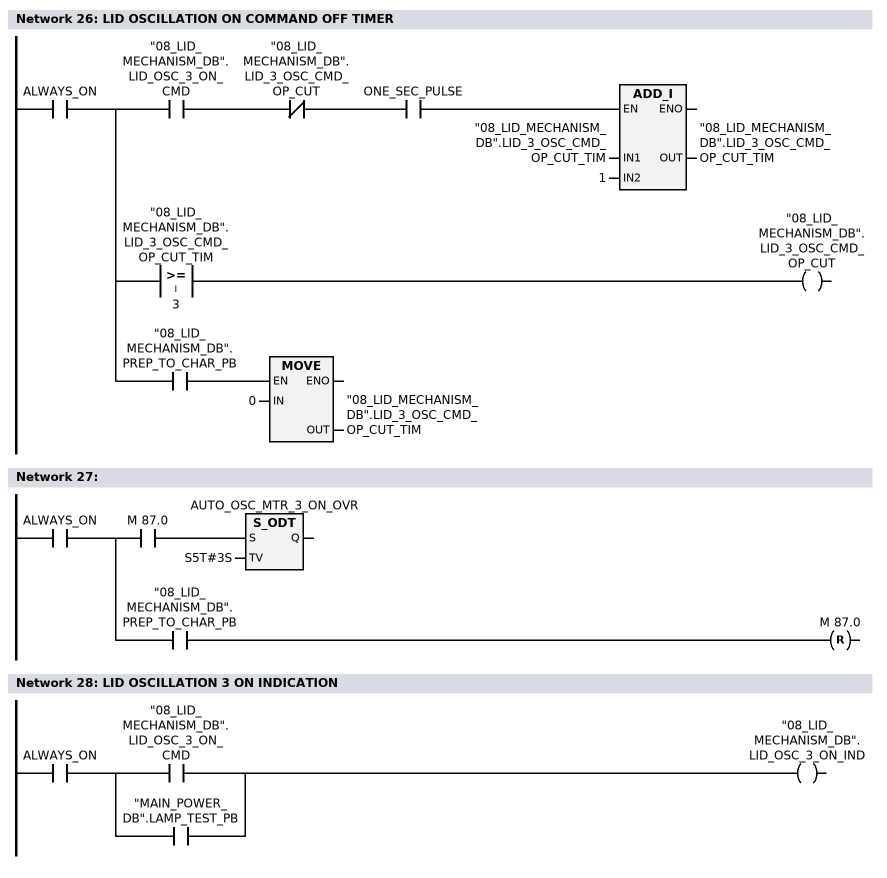
[picture p192: LID_3_MECHANISM networks 26-28]
NETWORK
TITLE = LID OSCILLATION ON COMMAND OFF TIMER
      A     "ALWAYS_ON";
      =     L 0.0;
      A     L 0.0;
      A     "08_LID_MECHANISM_DB".LID_OSC_3_ON_CMD;
      AN    "08_LID_MECHANISM_DB".LID_3_OSC_CMD_OP_CUT;
      A     "ONE_SEC_PULSE";
      JNB   _00d;
      L     "08_LID_MECHANISM_DB".LID_3_OSC_CMD_OP_CUT_TIM;
      L     1;
      +I;
      T     "08_LID_MECHANISM_DB".LID_3_OSC_CMD_OP_CUT_TIM;
_00d: NOP   0;
      A     L 0.0;
      A(;
      L     "08_LID_MECHANISM_DB".LID_3_OSC_CMD_OP_CUT_TIM;
      L     3;
      >=I;
      );
      =     "08_LID_MECHANISM_DB".LID_3_OSC_CMD_OP_CUT;
      A     L 0.0;
      A     "08_LID_MECHANISM_DB".PREP_TO_CHAR_PB;
      JNB   _00e;
      L     0;
      T     "08_LID_MECHANISM_DB".LID_3_OSC_CMD_OP_CUT_TIM;
_00e: NOP   0;
NETWORK
TITLE =
      A     "ALWAYS_ON";
      =     L 0.0;
      A     L 0.0;
      A     M 87.0;
      L     S5T#3S;
      SD    "AUTO_OSC_MTR_3_ON_OVR";
      NOP   0;
      NOP   0;
      NOP   0;
      NOP   0;
      A     L 0.0;
      A     "08_LID_MECHANISM_DB".PREP_TO_CHAR_PB;
      R     M 87.0;
NETWORK
TITLE = LID OSCILLATION 3 ON INDICATION
//CHECK IT
      A     "ALWAYS_ON";
      A(;
      O     "08_LID_MECHANISM_DB".LID_OSC_3_ON_CMD;
      O     "MAIN_POWER_DB".LAMP_TEST_PB;
      );
      =     "08_LID_MECHANISM_DB".LID_OSC_3_ON_IND;
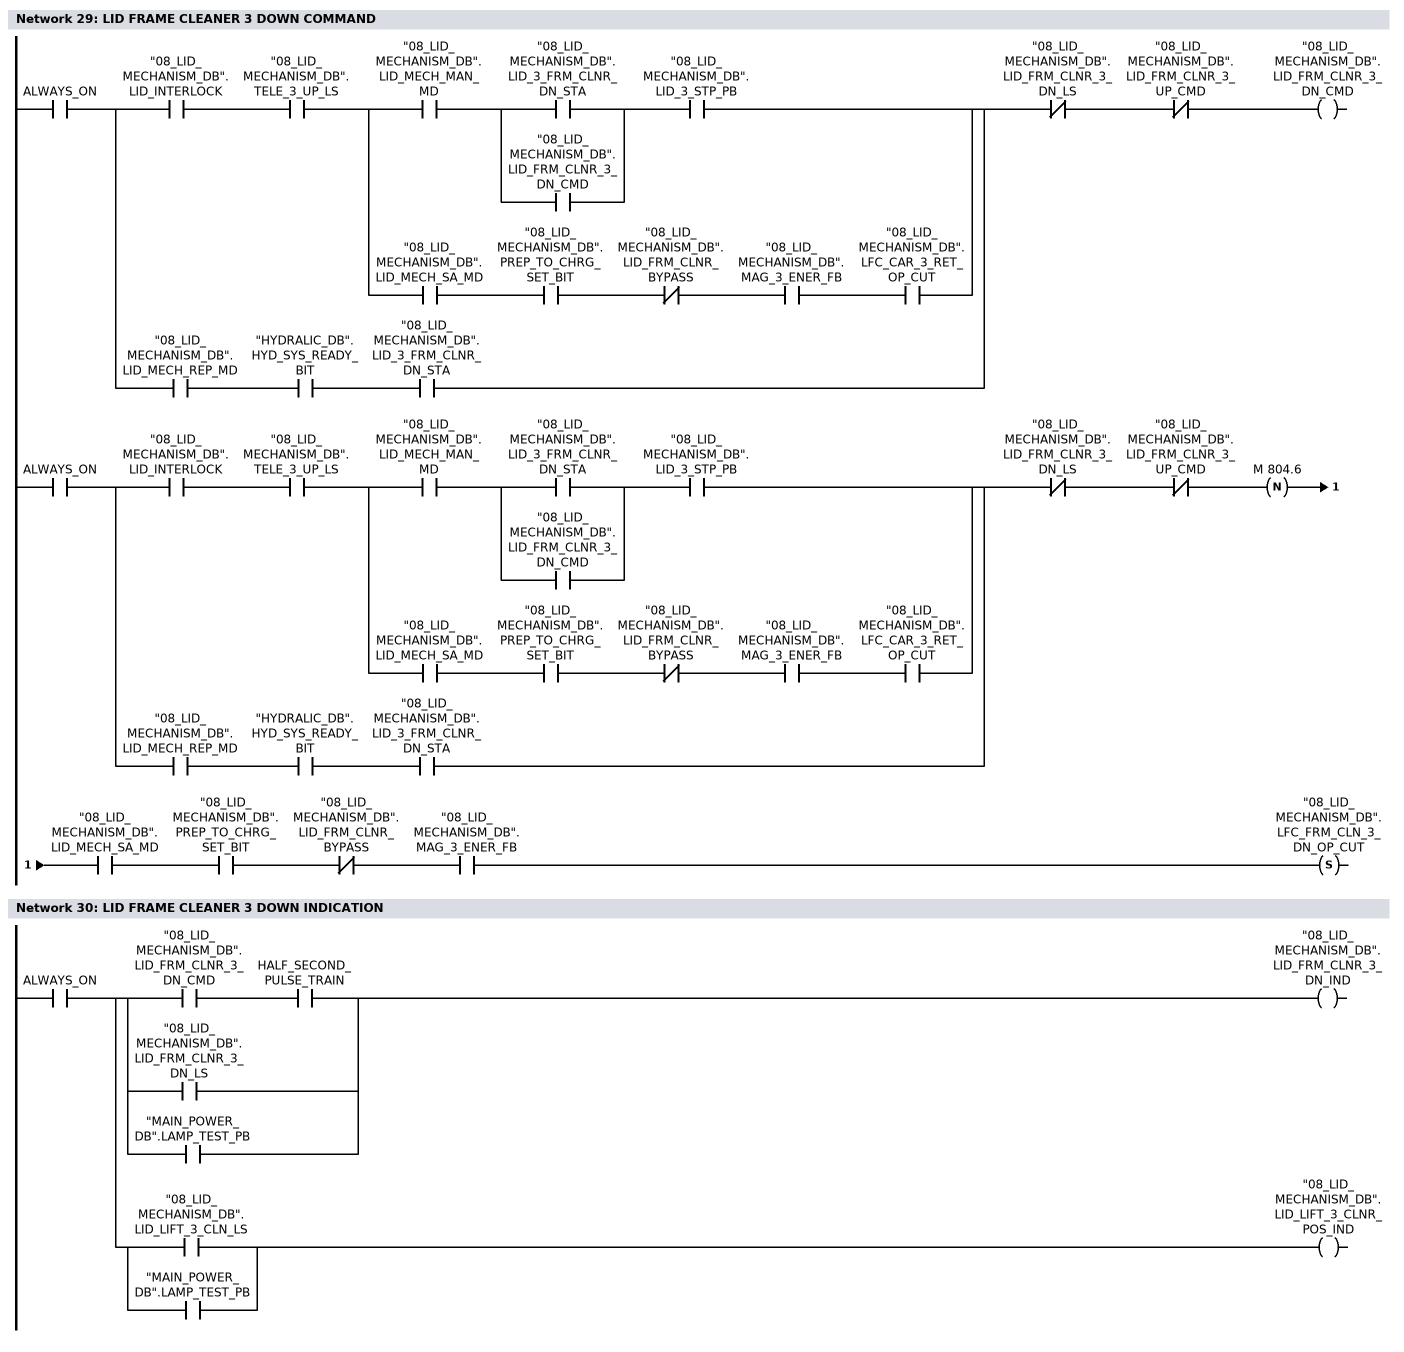
NETWORK
TITLE = LID FRAME CLEANER 3 DOWN COMMAND
      A     "ALWAYS_ON";
      A(;
      A     "08_LID_MECHANISM_DB".LID_INTERLOCK;
      A     "08_LID_MECHANISM_DB".TELE_3_UP_LS;
      A(;
      A     "08_LID_MECHANISM_DB".LID_MECH_MAN_MD;
      A(;
      O     "08_LID_MECHANISM_DB".LID_3_FRM_CLNR_DN_STA;
      O     "08_LID_MECHANISM_DB".LID_FRM_CLNR_3_DN_CMD;
      );
      A     "08_LID_MECHANISM_DB".LID_3_STP_PB;
      O;
      A     "08_LID_MECHANISM_DB".LID_MECH_SA_MD;
      A     "08_LID_MECHANISM_DB".PREP_TO_CHRG_SET_BIT;
      AN    "08_LID_MECHANISM_DB".LID_FRM_CLNR_BYPASS;
      A     "08_LID_MECHANISM_DB".MAG_3_ENER_FB;
      A     "08_LID_MECHANISM_DB".LFC_CAR_3_RET_OP_CUT;
      );
      O;
      A     "08_LID_MECHANISM_DB".LID_MECH_REP_MD;
      A     "HYDRALIC_DB".HYD_SYS_READY_BIT;
      A     "08_LID_MECHANISM_DB".LID_3_FRM_CLNR_DN_STA;
      );
      AN    "08_LID_MECHANISM_DB".LID_FRM_CLNR_3_DN_LS;
      AN    "08_LID_MECHANISM_DB".LID_FRM_CLNR_3_UP_CMD;
      =     L 0.0;
      A     L 0.0;
      BLD   102;
      =     "08_LID_MECHANISM_DB".LID_FRM_CLNR_3_DN_CMD;
      A(;
      A     L 0.0;
      FN    M 804.6;
      );
      A     "08_LID_MECHANISM_DB".LID_MECH_SA_MD;
      A     "08_LID_MECHANISM_DB".PREP_TO_CHRG_SET_BIT;
      AN    "08_LID_MECHANISM_DB".LID_FRM_CLNR_BYPASS;
      A     "08_LID_MECHANISM_DB".MAG_3_ENER_FB;
      S     "08_LID_MECHANISM_DB".LFC_FRM_CLN_3_DN_OP_CUT;
NETWORK
TITLE = LID FRAME CLEANER 3 DOWN INDICATION
      A     "ALWAYS_ON";
      =     L 0.0;
      A     L 0.0;
      A(;
      A     "08_LID_MECHANISM_DB".LID_FRM_CLNR_3_DN_CMD;
      A     "HALF_SECOND_PULSE_TRAIN";
      O     "08_LID_MECHANISM_DB".LID_FRM_CLNR_3_DN_LS;
      O     "MAIN_POWER_DB".LAMP_TEST_PB;
      );
      =     "08_LID_MECHANISM_DB".LID_FRM_CLNR_3_DN_IND;
      A     L 0.0;
      A(;
      O     "08_LID_MECHANISM_DB".LID_LIFT_3_CLN_LS;
      O     "MAIN_POWER_DB".LAMP_TEST_PB;
      );
      =     "08_LID_MECHANISM_DB".LID_LIFT_3_CLNR_POS_IND;
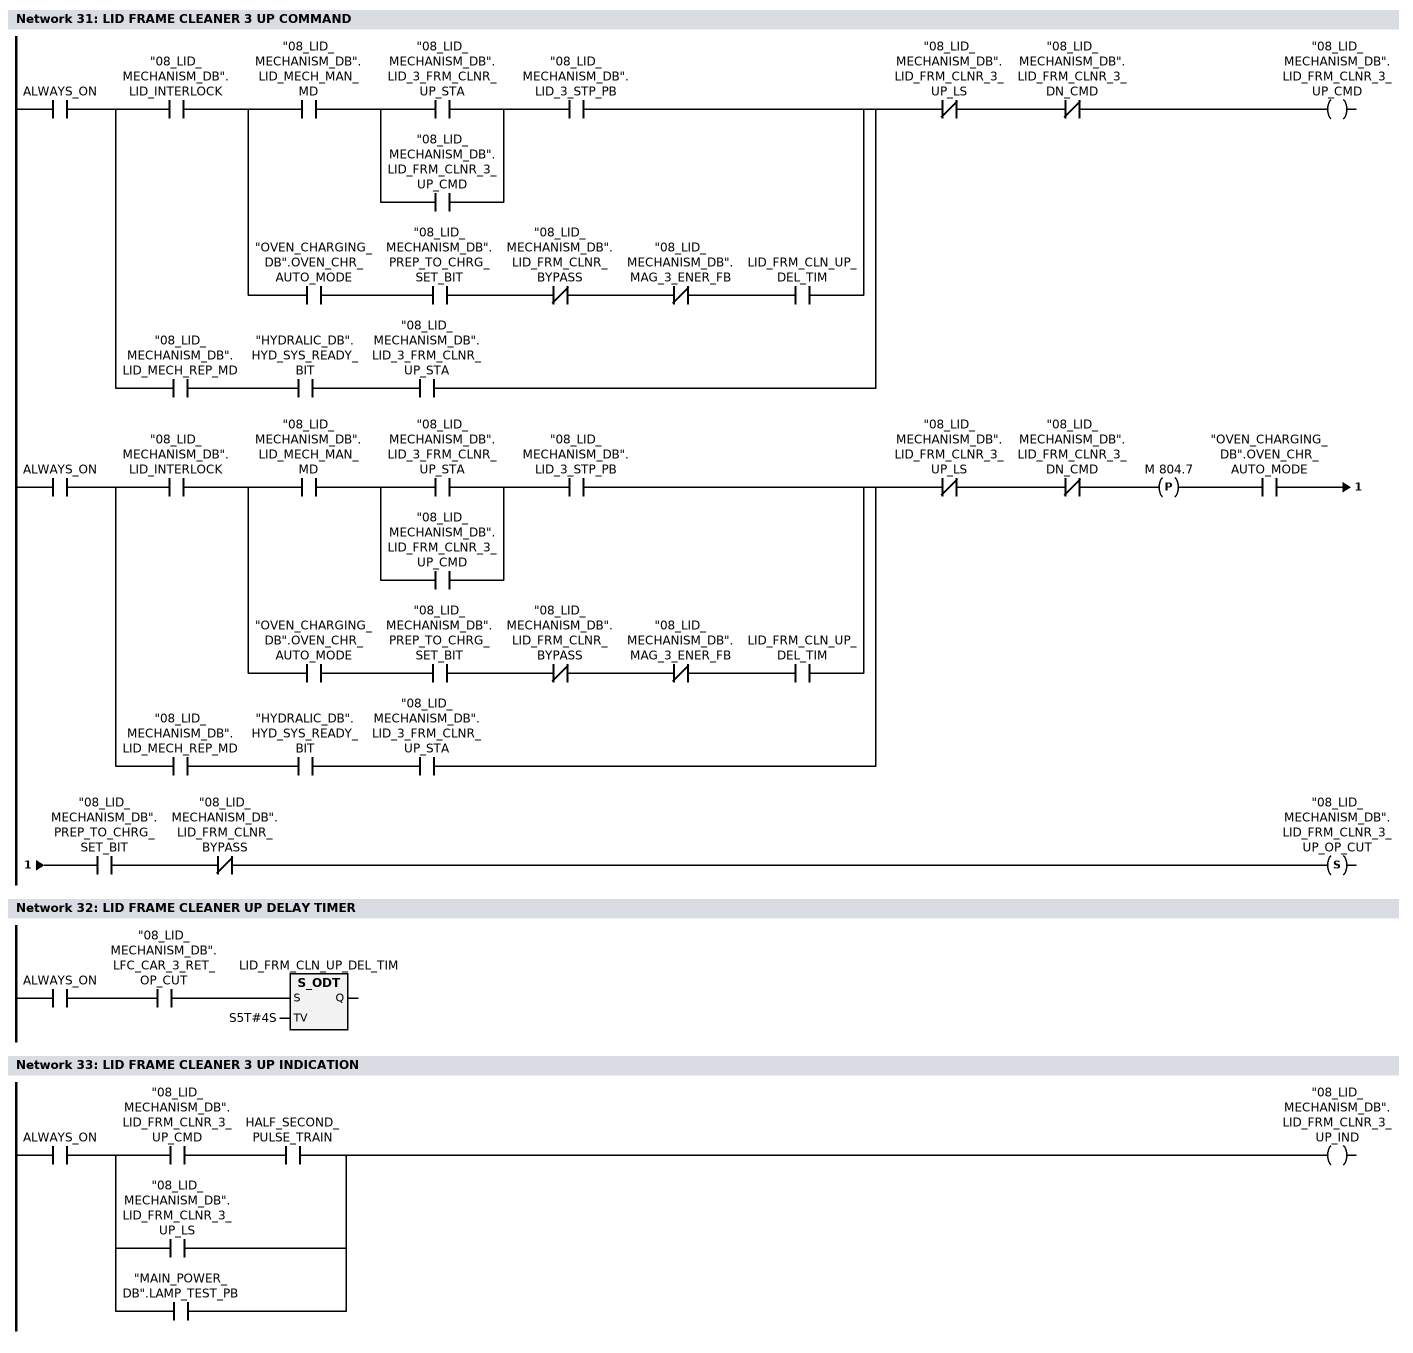
NETWORK
TITLE = LID FRAME CLEANER 3 UP COMMAND
      A     "ALWAYS_ON";
      A(;
      A     "08_LID_MECHANISM_DB".LID_INTERLOCK;
      A(;
      A     "08_LID_MECHANISM_DB".LID_MECH_MAN_MD;
      A(;
      O     "08_LID_MECHANISM_DB".LID_3_FRM_CLNR_UP_STA;
      O     "08_LID_MECHANISM_DB".LID_FRM_CLNR_3_UP_CMD;
      );
      A     "08_LID_MECHANISM_DB".LID_3_STP_PB;
      O;
      A     "OVEN_CHARGING_DB".OVEN_CHR_AUTO_MODE;
      A     "08_LID_MECHANISM_DB".PREP_TO_CHRG_SET_BIT;
      AN    "08_LID_MECHANISM_DB".LID_FRM_CLNR_BYPASS;
      AN    "08_LID_MECHANISM_DB".MAG_3_ENER_FB;
      A     "LID_FRM_CLN_UP_DEL_TIM";
      );
      O;
      A     "08_LID_MECHANISM_DB".LID_MECH_REP_MD;
      A     "HYDRALIC_DB".HYD_SYS_READY_BIT;
      A     "08_LID_MECHANISM_DB".LID_3_FRM_CLNR_UP_STA;
      );
      AN    "08_LID_MECHANISM_DB".LID_FRM_CLNR_3_UP_LS;
      AN    "08_LID_MECHANISM_DB".LID_FRM_CLNR_3_DN_CMD;
      =     L 0.0;
      A     L 0.0;
      BLD   102;
      =     "08_LID_MECHANISM_DB".LID_FRM_CLNR_3_UP_CMD;
      A(;
      A     L 0.0;
      FP    M 804.7;
      );
      A     "OVEN_CHARGING_DB".OVEN_CHR_AUTO_MODE;
      A     "08_LID_MECHANISM_DB".PREP_TO_CHRG_SET_BIT;
      AN    "08_LID_MECHANISM_DB".LID_FRM_CLNR_BYPASS;
      S     "08_LID_MECHANISM_DB".LID_FRM_CLNR_3_UP_OP_CUT;
NETWORK
TITLE = LID FRAME CLEANER UP DELAY TIMER
      A     "ALWAYS_ON";
      A     "08_LID_MECHANISM_DB".LFC_CAR_3_RET_OP_CUT;
      L     S5T#4S;
      SD    "LID_FRM_CLN_UP_DEL_TIM";
      NOP   0;
      NOP   0;
      NOP   0;
      NOP   0;
NETWORK
TITLE = LID FRAME CLEANER 3 UP INDICATION
      A     "ALWAYS_ON";
      A(;
      A     "08_LID_MECHANISM_DB".LID_FRM_CLNR_3_UP_CMD;
      A     "HALF_SECOND_PULSE_TRAIN";
      O     "08_LID_MECHANISM_DB".LID_FRM_CLNR_3_UP_LS;
      O     "MAIN_POWER_DB".LAMP_TEST_PB;
      );
      =     "08_LID_MECHANISM_DB".LID_FRM_CLNR_3_UP_IND;
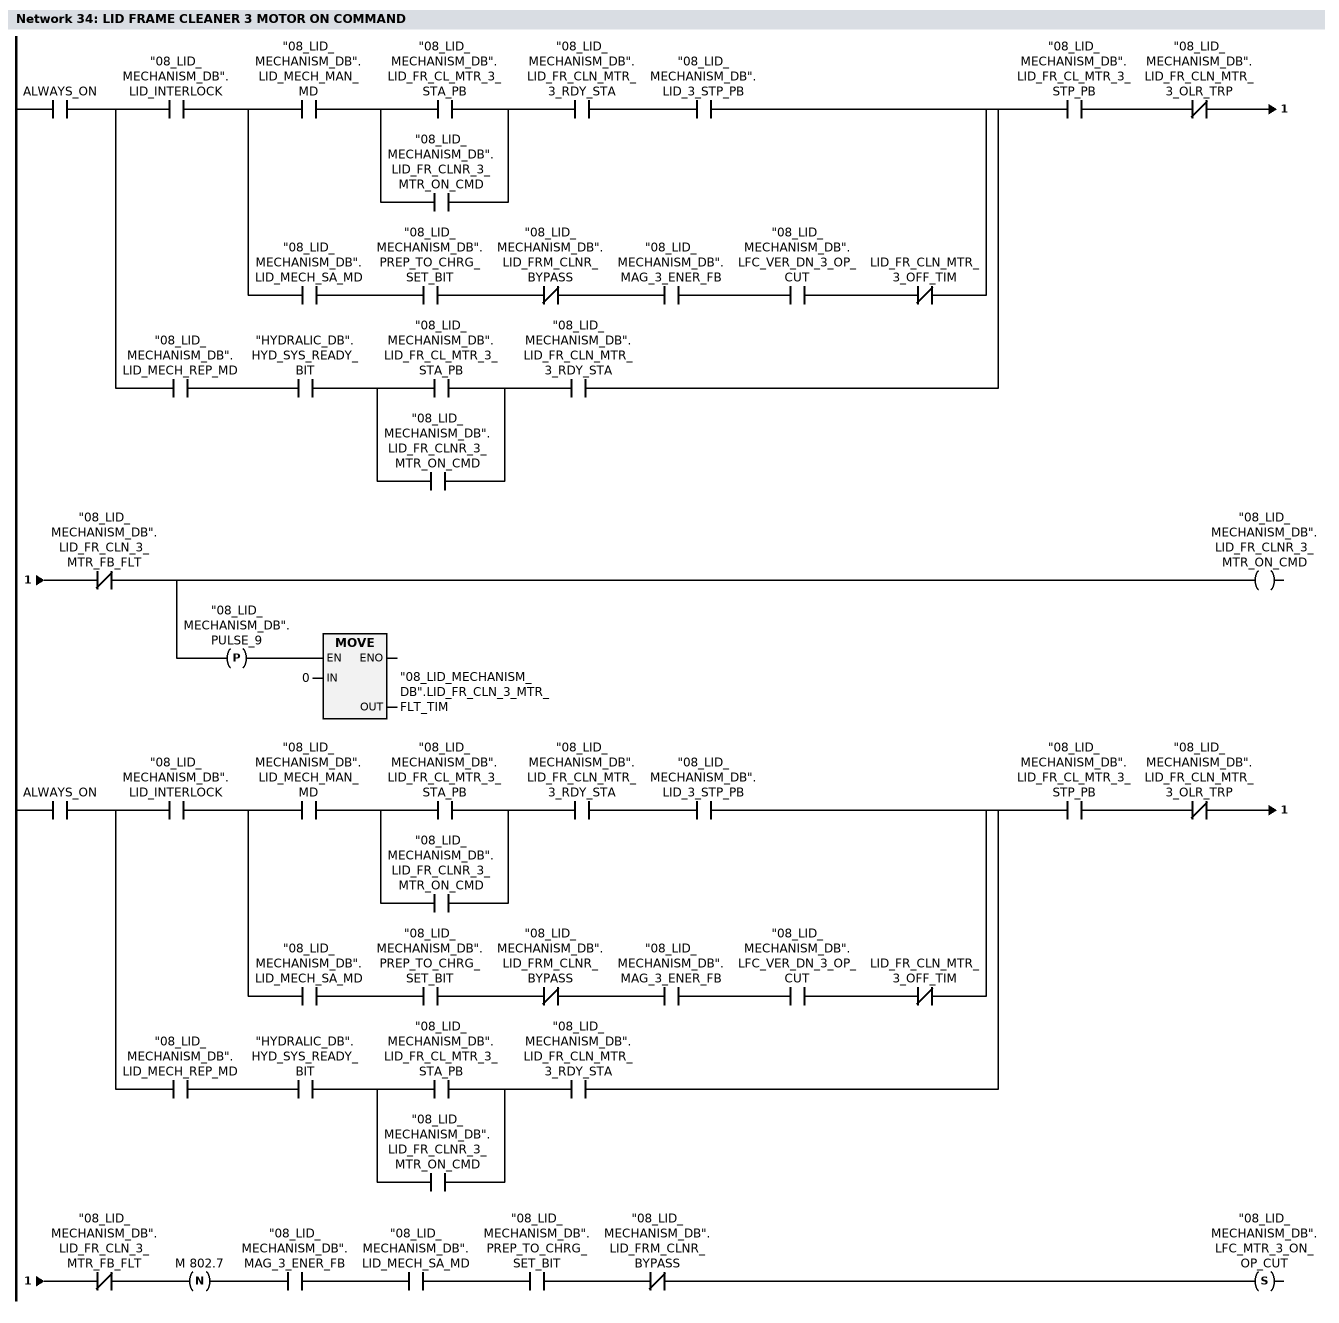
NETWORK
TITLE = LID FRAME CLEANER 3 MOTOR ON COMMAND
      A     "ALWAYS_ON";
      A(;
      A     "08_LID_MECHANISM_DB".LID_INTERLOCK;
      A(;
      A     "08_LID_MECHANISM_DB".LID_MECH_MAN_MD;
      A(;
      O     "08_LID_MECHANISM_DB".LID_FR_CL_MTR_3_STA_PB;
      O     "08_LID_MECHANISM_DB".LID_FR_CLNR_3_MTR_ON_CMD;
      );
      A     "08_LID_MECHANISM_DB".LID_FR_CLN_MTR_3_RDY_STA;
      A     "08_LID_MECHANISM_DB".LID_3_STP_PB;
      O;
      A     "08_LID_MECHANISM_DB".LID_MECH_SA_MD;
      A     "08_LID_MECHANISM_DB".PREP_TO_CHRG_SET_BIT;
      AN    "08_LID_MECHANISM_DB".LID_FRM_CLNR_BYPASS;
      A     "08_LID_MECHANISM_DB".MAG_3_ENER_FB;
      A     "08_LID_MECHANISM_DB".LFC_VER_DN_3_OP_CUT;
      AN    "LID_FR_CLN_MTR_3_OFF_TIM";
      );
      O;
      A     "08_LID_MECHANISM_DB".LID_MECH_REP_MD;
      A     "HYDRALIC_DB".HYD_SYS_READY_BIT;
      A(;
      O     "08_LID_MECHANISM_DB".LID_FR_CL_MTR_3_STA_PB;
      O     "08_LID_MECHANISM_DB".LID_FR_CLNR_3_MTR_ON_CMD;
      );
      A     "08_LID_MECHANISM_DB".LID_FR_CLN_MTR_3_RDY_STA;
      );
      A     "08_LID_MECHANISM_DB".LID_FR_CL_MTR_3_STP_PB;
      AN    "08_LID_MECHANISM_DB".LID_FR_CLN_MTR_3_OLR_TRP;
      AN    "08_LID_MECHANISM_DB".LID_FR_CLN_3_MTR_FB_FLT;
      =     L 0.0;
      A     L 0.0;
      BLD   102;
      =     "08_LID_MECHANISM_DB".LID_FR_CLNR_3_MTR_ON_CMD;
      A     L 0.0;
      FP    "08_LID_MECHANISM_DB".PULSE_9;
      JNB   _00f;
      L     0;
      T     "08_LID_MECHANISM_DB".LID_FR_CLN_3_MTR_FLT_TIM;
_00f: NOP   0;
      A(;
      A     L 0.0;
      FN    M 802.7;
      );
      A     "08_LID_MECHANISM_DB".MAG_3_ENER_FB;
      A     "08_LID_MECHANISM_DB".LID_MECH_SA_MD;
      A     "08_LID_MECHANISM_DB".PREP_TO_CHRG_SET_BIT;
      AN    "08_LID_MECHANISM_DB".LID_FRM_CLNR_BYPASS;
      S     "08_LID_MECHANISM_DB".LFC_MTR_3_ON_OP_CUT;
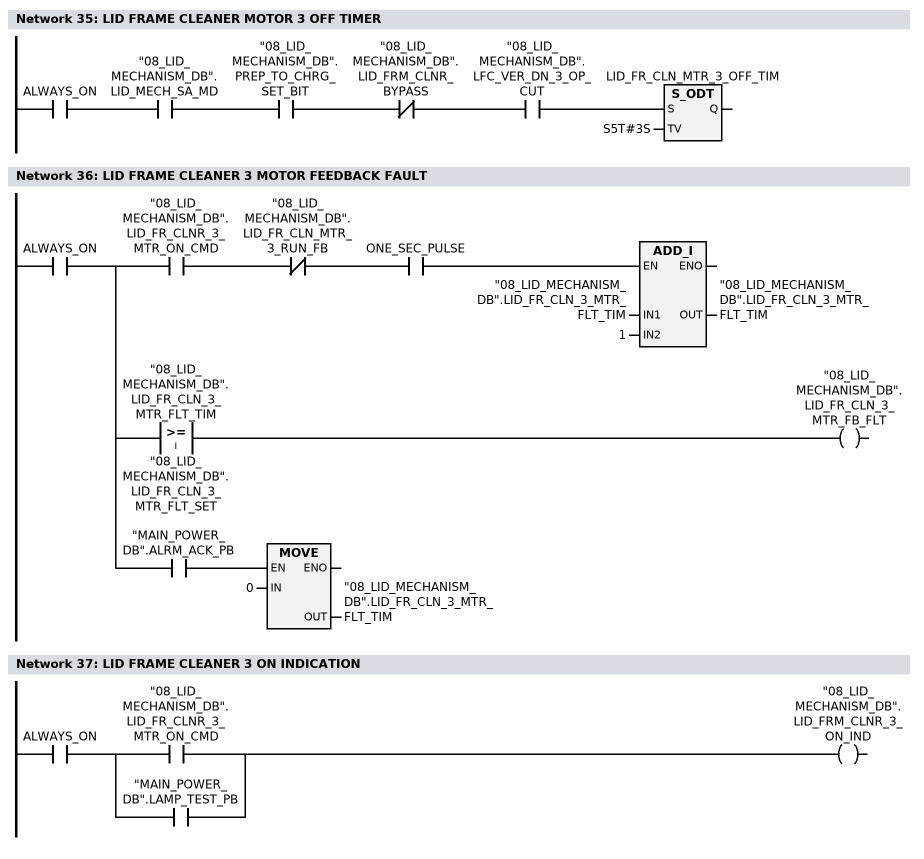
NETWORK
TITLE = LID FRAME CLEANER MOTOR 3 OFF TIMER
      A     "ALWAYS_ON";
      A     "08_LID_MECHANISM_DB".LID_MECH_SA_MD;
      A     "08_LID_MECHANISM_DB".PREP_TO_CHRG_SET_BIT;
      AN    "08_LID_MECHANISM_DB".LID_FRM_CLNR_BYPASS;
      A     "08_LID_MECHANISM_DB".LFC_VER_DN_3_OP_CUT;
      L     S5T#3S;
      SD    "LID_FR_CLN_MTR_3_OFF_TIM";
      NOP   0;
      NOP   0;
      NOP   0;
      NOP   0;
NETWORK
TITLE = LID FRAME CLEANER 3 MOTOR FEEDBACK FAULT
      A     "ALWAYS_ON";
      =     L 0.0;
      A     L 0.0;
      A     "08_LID_MECHANISM_DB".LID_FR_CLNR_3_MTR_ON_CMD;
      AN    "08_LID_MECHANISM_DB".LID_FR_CLN_MTR_3_RUN_FB;
      A     "ONE_SEC_PULSE";
      JNB   _010;
      L     "08_LID_MECHANISM_DB".LID_FR_CLN_3_MTR_FLT_TIM;
      L     1;
      +I;
      T     "08_LID_MECHANISM_DB".LID_FR_CLN_3_MTR_FLT_TIM;
_010: NOP   0;
      A     L 0.0;
      A(;
      L     "08_LID_MECHANISM_DB".LID_FR_CLN_3_MTR_FLT_TIM;
      L     "08_LID_MECHANISM_DB".LID_FR_CLN_3_MTR_FLT_SET;
      >=I;
      );
      =     "08_LID_MECHANISM_DB".LID_FR_CLN_3_MTR_FB_FLT;
      A     L 0.0;
      A     "MAIN_POWER_DB".ALRM_ACK_PB;
      JNB   _011;
      L     0;
      T     "08_LID_MECHANISM_DB".LID_FR_CLN_3_MTR_FLT_TIM;
_011: NOP   0;
NETWORK
TITLE = LID FRAME CLEANER 3 ON INDICATION
      A     "ALWAYS_ON";
      A(;
      O     "08_LID_MECHANISM_DB".LID_FR_CLNR_3_MTR_ON_CMD;
      O     "MAIN_POWER_DB".LAMP_TEST_PB;
      );
      =     "08_LID_MECHANISM_DB".LID_FRM_CLNR_3_ON_IND;
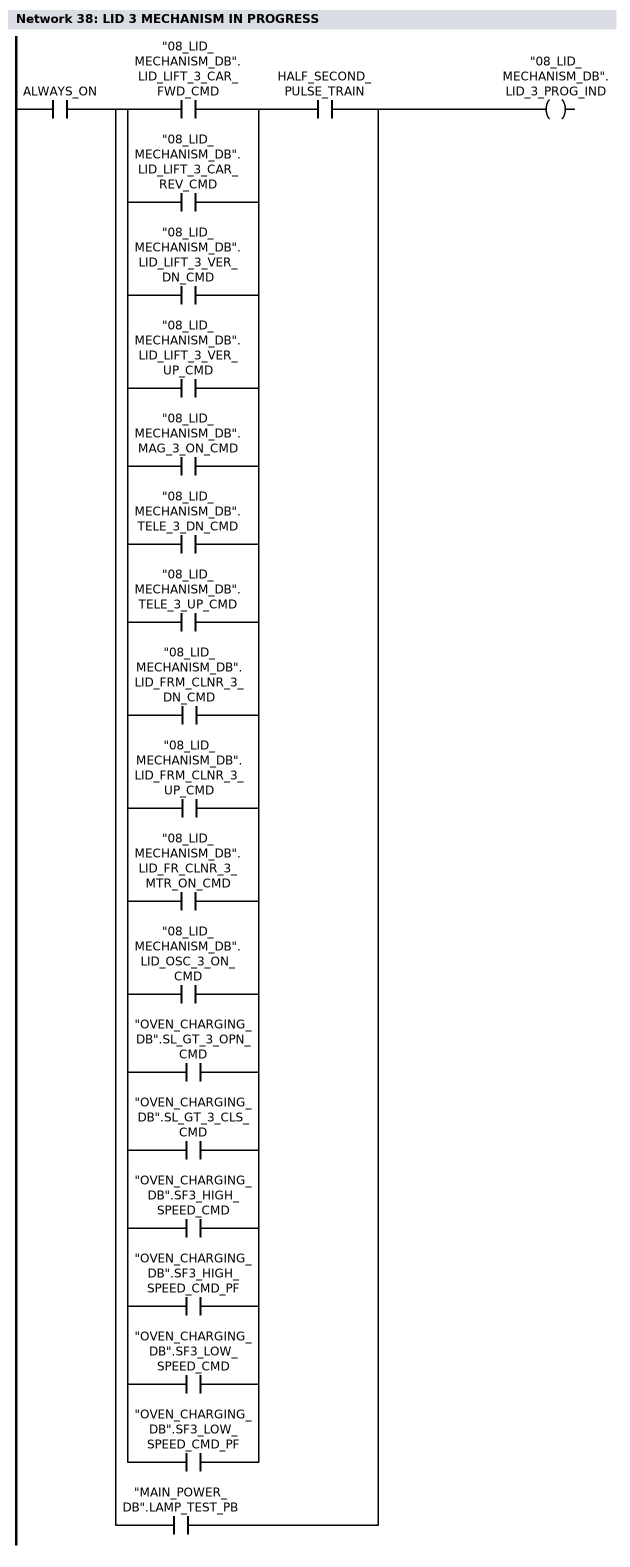
NETWORK
TITLE = LID 3 MECHANISM IN PROGRESS
      A     "ALWAYS_ON";
      A(;
      A(;
      O     "08_LID_MECHANISM_DB".LID_LIFT_3_CAR_FWD_CMD;
      O     "08_LID_MECHANISM_DB".LID_LIFT_3_CAR_REV_CMD;
      O     "08_LID_MECHANISM_DB".LID_LIFT_3_VER_DN_CMD;
      O     "08_LID_MECHANISM_DB".LID_LIFT_3_VER_UP_CMD;
      O     "08_LID_MECHANISM_DB".MAG_3_ON_CMD;
      O     "08_LID_MECHANISM_DB".TELE_3_DN_CMD;
      O     "08_LID_MECHANISM_DB".TELE_3_UP_CMD;
      O     "08_LID_MECHANISM_DB".LID_FRM_CLNR_3_DN_CMD;
      O     "08_LID_MECHANISM_DB".LID_FRM_CLNR_3_UP_CMD;
      O     "08_LID_MECHANISM_DB".LID_FR_CLNR_3_MTR_ON_CMD;
      O     "08_LID_MECHANISM_DB".LID_OSC_3_ON_CMD;
      O     "OVEN_CHARGING_DB".SL_GT_3_OPN_CMD;
      O     "OVEN_CHARGING_DB".SL_GT_3_CLS_CMD;
      O     "OVEN_CHARGING_DB".SF3_HIGH_SPEED_CMD;
      O     "OVEN_CHARGING_DB".SF3_HIGH_SPEED_CMD_PF;
      O     "OVEN_CHARGING_DB".SF3_LOW_SPEED_CMD;
      O     "OVEN_CHARGING_DB".SF3_LOW_SPEED_CMD_PF;
      );
      A     "HALF_SECOND_PULSE_TRAIN";
      O     "MAIN_POWER_DB".LAMP_TEST_PB;
      );
      =     "08_LID_MECHANISM_DB".LID_3_PROG_IND;
END_FUNCTION

FUNCTION "TATA_COMMUNICATION" : VOID	// FC 21
AUTHOR : Arun
VERSION : 0.1
BEGIN
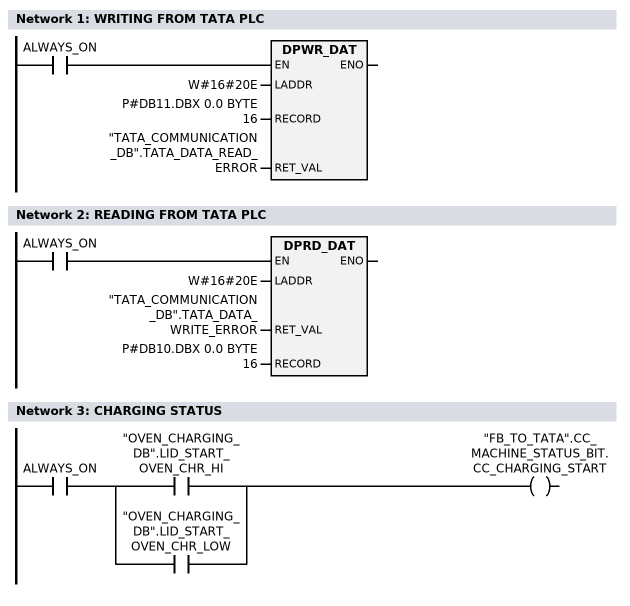
NETWORK
TITLE = WRITING FROM TATA PLC
      A     "ALWAYS_ON";
      JNB   _001;
      CALL  "DPWR_DAT" (
           LADDR                    := W#16#20E,
           RECORD                   := P#DB11.DBX 0.0 BYTE 16,
           RET_VAL                  := "TATA_COMMUNICATION_DB".TATA_DATA_READ_ERROR);
_001: NOP   0;
NETWORK
TITLE = READING FROM TATA PLC
      A     "ALWAYS_ON";
      JNB   _002;
      CALL  "DPRD_DAT" (
           LADDR                    := W#16#20E,
           RET_VAL                  := "TATA_COMMUNICATION_DB".TATA_DATA_WRITE_ERROR,
           RECORD                   := P#DB10.DBX 0.0 BYTE 16);
_002: NOP   0;
NETWORK
TITLE = CHARGING STATUS
      A     "ALWAYS_ON";
      A(;
      O     "OVEN_CHARGING_DB".LID_START_OVEN_CHR_HI;
      O     "OVEN_CHARGING_DB".LID_START_OVEN_CHR_LOW;
      );
      =     "FB_TO_TATA".CC_MACHINE_STATUS_BIT.CC_CHARGING_START;
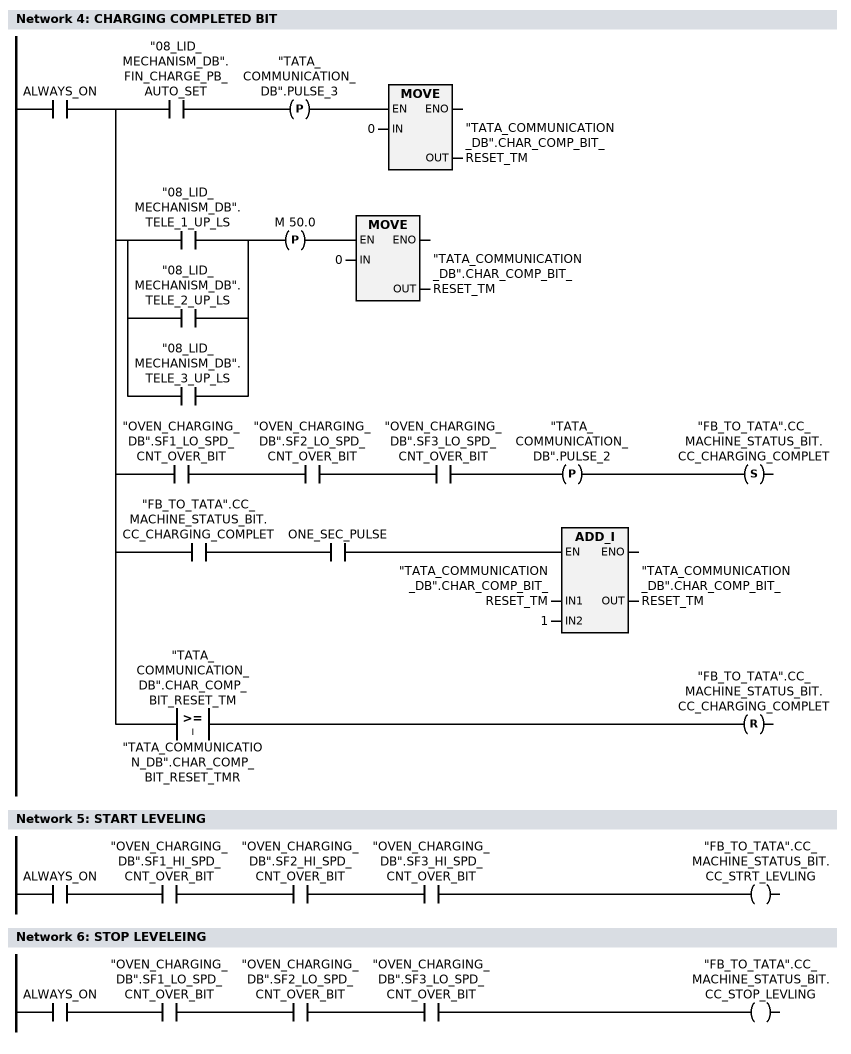
NETWORK
TITLE = CHARGING COMPLETED BIT
      A     "ALWAYS_ON";
      =     L 0.0;
      A     L 0.0;
      A     "08_LID_MECHANISM_DB".FIN_CHARGE_PB_AUTO_SET;
      FP    "TATA_COMMUNICATION_DB".PULSE_3;
      JNB   _003;
      L     0;
      T     "TATA_COMMUNICATION_DB".CHAR_COMP_BIT_RESET_TM;
_003: NOP   0;
      A     L 0.0;
      A(;
      O     "08_LID_MECHANISM_DB".TELE_1_UP_LS;
      O     "08_LID_MECHANISM_DB".TELE_2_UP_LS;
      O     "08_LID_MECHANISM_DB".TELE_3_UP_LS;
      );
      FP    M 50.0;
      JNB   _004;
      L     0;
      T     "TATA_COMMUNICATION_DB".CHAR_COMP_BIT_RESET_TM;
_004: NOP   0;
      A     L 0.0;
      A     "OVEN_CHARGING_DB".SF1_LO_SPD_CNT_OVER_BIT;
      A     "OVEN_CHARGING_DB".SF2_LO_SPD_CNT_OVER_BIT;
      A     "OVEN_CHARGING_DB".SF3_LO_SPD_CNT_OVER_BIT;
      FP    "TATA_COMMUNICATION_DB".PULSE_2;
      S     "FB_TO_TATA".CC_MACHINE_STATUS_BIT.CC_CHARGING_COMPLET;
      A     L 0.0;
      A     "FB_TO_TATA".CC_MACHINE_STATUS_BIT.CC_CHARGING_COMPLET;
      A     "ONE_SEC_PULSE";
      JNB   _005;
      L     "TATA_COMMUNICATION_DB".CHAR_COMP_BIT_RESET_TM;
      L     1;
      +I;
      T     "TATA_COMMUNICATION_DB".CHAR_COMP_BIT_RESET_TM;
_005: NOP   0;
      A     L 0.0;
      A(;
      L     "TATA_COMMUNICATION_DB".CHAR_COMP_BIT_RESET_TM;
      L     "TATA_COMMUNICATION_DB".CHAR_COMP_BIT_RESET_TMR;
      >=I;
      );
      R     "FB_TO_TATA".CC_MACHINE_STATUS_BIT.CC_CHARGING_COMPLET;
NETWORK
TITLE = START LEVELING
      A     "ALWAYS_ON";
      A     "OVEN_CHARGING_DB".SF1_HI_SPD_CNT_OVER_BIT;
      A     "OVEN_CHARGING_DB".SF2_HI_SPD_CNT_OVER_BIT;
      A     "OVEN_CHARGING_DB".SF3_HI_SPD_CNT_OVER_BIT;
      =     "FB_TO_TATA".CC_MACHINE_STATUS_BIT.CC_STRT_LEVLING;
NETWORK
TITLE = STOP LEVELEING
      A     "ALWAYS_ON";
      A     "OVEN_CHARGING_DB".SF1_LO_SPD_CNT_OVER_BIT;
      A     "OVEN_CHARGING_DB".SF2_LO_SPD_CNT_OVER_BIT;
      A     "OVEN_CHARGING_DB".SF3_LO_SPD_CNT_OVER_BIT;
      =     "FB_TO_TATA".CC_MACHINE_STATUS_BIT.CC_STOP_LEVLING;
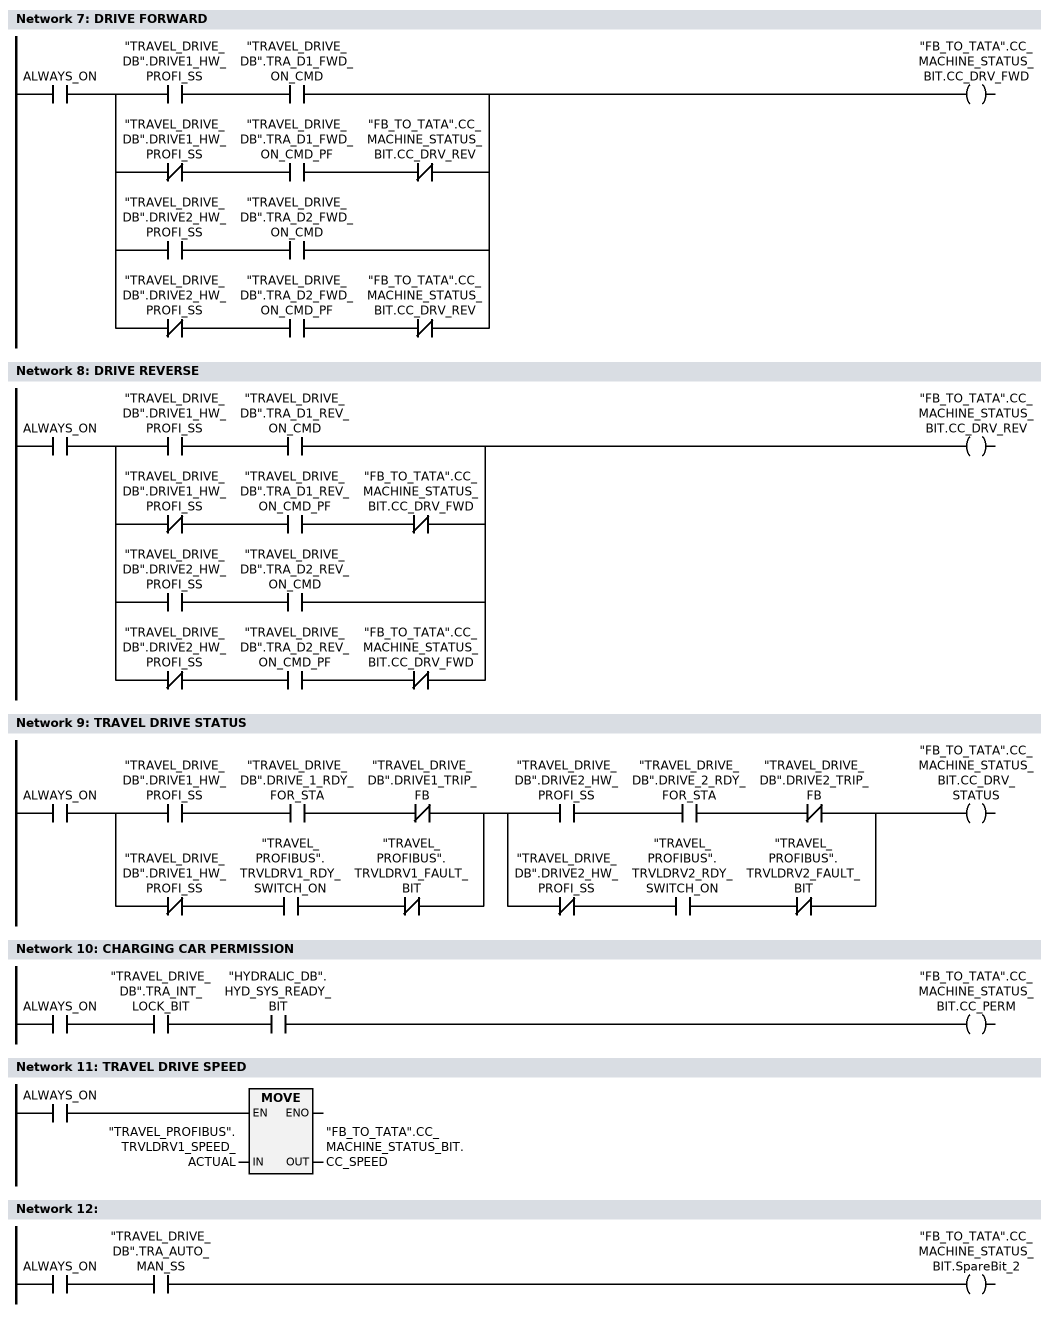
NETWORK
TITLE = DRIVE FORWARD
      A     "ALWAYS_ON";
      A(;
      A     "TRAVEL_DRIVE_DB".DRIVE1_HW_PROFI_SS;
      A     "TRAVEL_DRIVE_DB".TRA_D1_FWD_ON_CMD;
      O;
      AN    "TRAVEL_DRIVE_DB".DRIVE1_HW_PROFI_SS;
      A     "TRAVEL_DRIVE_DB".TRA_D1_FWD_ON_CMD_PF;
      AN    "FB_TO_TATA".CC_MACHINE_STATUS_BIT.CC_DRV_REV;
      O;
      A     "TRAVEL_DRIVE_DB".DRIVE2_HW_PROFI_SS;
      A     "TRAVEL_DRIVE_DB".TRA_D2_FWD_ON_CMD;
      O;
      AN    "TRAVEL_DRIVE_DB".DRIVE2_HW_PROFI_SS;
      A     "TRAVEL_DRIVE_DB".TRA_D2_FWD_ON_CMD_PF;
      AN    "FB_TO_TATA".CC_MACHINE_STATUS_BIT.CC_DRV_REV;
      );
      =     "FB_TO_TATA".CC_MACHINE_STATUS_BIT.CC_DRV_FWD;
NETWORK
TITLE = DRIVE REVERSE
      A     "ALWAYS_ON";
      A(;
      A     "TRAVEL_DRIVE_DB".DRIVE1_HW_PROFI_SS;
      A     "TRAVEL_DRIVE_DB".TRA_D1_REV_ON_CMD;
      O;
      AN    "TRAVEL_DRIVE_DB".DRIVE1_HW_PROFI_SS;
      A     "TRAVEL_DRIVE_DB".TRA_D1_REV_ON_CMD_PF;
      AN    "FB_TO_TATA".CC_MACHINE_STATUS_BIT.CC_DRV_FWD;
      O;
      A     "TRAVEL_DRIVE_DB".DRIVE2_HW_PROFI_SS;
      A     "TRAVEL_DRIVE_DB".TRA_D2_REV_ON_CMD;
      O;
      AN    "TRAVEL_DRIVE_DB".DRIVE2_HW_PROFI_SS;
      A     "TRAVEL_DRIVE_DB".TRA_D2_REV_ON_CMD_PF;
      AN    "FB_TO_TATA".CC_MACHINE_STATUS_BIT.CC_DRV_FWD;
      );
      =     "FB_TO_TATA".CC_MACHINE_STATUS_BIT.CC_DRV_REV;
NETWORK
TITLE = TRAVEL DRIVE STATUS
      A     "ALWAYS_ON";
      A(;
      A     "TRAVEL_DRIVE_DB".DRIVE1_HW_PROFI_SS;
      A     "TRAVEL_DRIVE_DB".DRIVE_1_RDY_FOR_STA;
      AN    "TRAVEL_DRIVE_DB".DRIVE1_TRIP_FB;
      O;
      AN    "TRAVEL_DRIVE_DB".DRIVE1_HW_PROFI_SS;
      A     "TRAVEL_PROFIBUS".TRVLDRV1_RDY_SWITCH_ON;
      AN    "TRAVEL_PROFIBUS".TRVLDRV1_FAULT_BIT;
      );
      A(;
      A     "TRAVEL_DRIVE_DB".DRIVE2_HW_PROFI_SS;
      A     "TRAVEL_DRIVE_DB".DRIVE_2_RDY_FOR_STA;
      AN    "TRAVEL_DRIVE_DB".DRIVE2_TRIP_FB;
      O;
      AN    "TRAVEL_DRIVE_DB".DRIVE2_HW_PROFI_SS;
      A     "TRAVEL_PROFIBUS".TRVLDRV2_RDY_SWITCH_ON;
      AN    "TRAVEL_PROFIBUS".TRVLDRV2_FAULT_BIT;
      );
      =     "FB_TO_TATA".CC_MACHINE_STATUS_BIT.CC_DRV_STATUS;
NETWORK
TITLE = CHARGING CAR PERMISSION
      A     "ALWAYS_ON";
      A     "TRAVEL_DRIVE_DB".TRA_INT_LOCK_BIT;
      A     "HYDRALIC_DB".HYD_SYS_READY_BIT;
      =     "FB_TO_TATA".CC_MACHINE_STATUS_BIT.CC_PERM;
NETWORK
TITLE = TRAVEL DRIVE SPEED
      A     "ALWAYS_ON";
      JNB   _006;
      L     "TRAVEL_PROFIBUS".TRVLDRV1_SPEED_ACTUAL;
      T     "FB_TO_TATA".CC_MACHINE_STATUS_BIT.CC_SPEED;
_006: NOP   0;
NETWORK
TITLE =
      A     "ALWAYS_ON";
      A     "TRAVEL_DRIVE_DB".TRA_AUTO_MAN_SS;
      =     "FB_TO_TATA".CC_MACHINE_STATUS_BIT.SpareBit_2;
END_FUNCTION

// FC 105: know-how protected block, not included

// FC 106: know-how protected block, not included

DATA_BLOCK "MAIN_POWER_DB"	// DB 1
VERSION : 0.1
  STRUCT
   MAIN_PWR_RDY_FOR_ON : BOOL ;	//MAIN POWER READY FOR ON
   MAIN_PWR_RUN_FB : BOOL ;	//MAIN POWER ON FEEDBACK
   CTRL_PWR_ON_FB : BOOL ;	//CONTROL POWER ON FEEDBACK
   MAIN_PWR_ON_PB : BOOL ;	//MAIN POWER ON PUSH BUTTON
   MAIN_PWR_OFF_PB : BOOL ;	//MAIN POWER OFF PUSH BUTTON
   LAMP_TEST_PB : BOOL ;	//MAIN POWER LAMP TEST PUSH BUTTON
   ALRM_ACK_PB : BOOL ;	//MAIN POWER ALARM ACKNOWLEDGE PUSH BUTTON
   MAIN_PWR_ON_CMD : BOOL ;	//MAIN POWER ON COMMAND
   MAIN_PWR_ON_IND : BOOL ;	//MAIN POWER ON INDICATION
   CTRL_PWR_ON_IND : BOOL ;	//CONTROL POWER ON INDICATION
   LIMIT_SWITCH_END_FWD_FB : BOOL ;	//LIMIT SWITCH TO CONTROL OVER TRAVEL
   MAIN_PWR_FB_TMR_SET : INT ;
   MAIN_PWR_FB_TMR_TIME : INT ;
   CTRL_PWR_FB_TMR_SET : INT ;
   CTRL_PWR_FB_TMR_TIME : INT ;
   MAIN_PWR_FB_FLT : BOOL ;	//MAIN POWER FEEDBACK FAILED
   CTRL_PWR_FB_FLT : BOOL ;	//CONTROL POWER FEEDBACK FAILED
   MAIN_PWR_HEALTHY : BOOL ;	//MAIN POWER HEALTHY BIT
  END_STRUCT ;	
BEGIN
   MAIN_PWR_FB_TMR_SET := 5;
   CTRL_PWR_FB_TMR_SET := 5;
END_DATA_BLOCK

DATA_BLOCK "HYDRALIC_DB"	// DB 2
VERSION : 0.1
  STRUCT
   HYD_PUMP1_RDY_FOR_STA : BOOL ;	//HYDRALIC PUMP1 READY FOR START
   HYD_PUMP1_RUN_FB : BOOL ;	//HYDRALIC PUMP1 RUNNING FEED BACK
   HYD_PUMP1_OLR : BOOL ;	//HYDRALIC PUMP1 OVER LOAD TRIP
   HYD_PUMP2_RDY_FOR_STA : BOOL ;	//HYDRALIC PUMP2 READY FOR START
   HYD_PUMP2_RUN_FB : BOOL ;	//HYDRALIC PUMP2 RUNNING FEED BACK
   HYD_PUMP2_OLR : BOOL ;	//HYDRALIC PUMP2 OVER LOAD TRIP
   CIR_PUMP_RDY_FOR_STA : BOOL ;	//CIRCULATION PUMP READY FOR START
   CIR_PUMP_RUN_FB : BOOL ;	//CIRCULATION PUMP RUNNING FEED BACK
   CIR_PUMP1_OLR : BOOL ;	//CIRCULATION PUMP OVER LOAD TRIP
   COOL_FAN_RDY_FOR_STA : BOOL ;	//COOLING FAN READY FOR START
   COOL_FAN_RUN_FB : BOOL ;	//COOLING FAN RUNNING FEED BACK
   COOL_FAN_OLR : BOOL ;	//COOLING FAN OVER LOAD TRIP
   HYD_CD_OR_LCS_SS : BOOL ;	//HYDRALIC CONTROLDESK OR LCS SELECTOR SWITCH
   PUMP_1OR2_SS : BOOL ;	//PUMP 1 OR 2 SELECTOR SWITCH
   PUMP1_STA_PB : BOOL ;	//PUMP1 START PUSH BUTTON
   PUMP1_STP_PB : BOOL ;	//PUMP1 STOP PUSH BUTTON
   PUMP2_STA_PB : BOOL ;	//PUMP2 START PUSH BUTTON
   PUMP2_STP_PB : BOOL ;	//PUMP2 STOP PUSH BUTTON
   EM_PB_LCS : BOOL ;	//EMERGENCY PUSH BUTTON LCS
   PUMP_1OR2_SS_LCS : BOOL ;	//PUMP 1 OR 2 SELECTOR SWITCH LCS
   PUMP1_STA_PB_LCS : BOOL ;	//PUMP1 START PUSH BUTTON LCS
   PUMP1_STP_PB_LCS : BOOL ;	//PUMP1 STOP PUSH BUTTON LCS
   PUMP2_STA_PB_LCS : BOOL ;	//PUMP2 START PUSH BUTTON LCS
   PUMP2_STP_PB_LCS : BOOL ;	//PUMP2 STOP PUSH BUTTON LCS
   CIR_PUMP_STA_PB : BOOL ;	//CIRCULATION PUMP START PUSH BUTTON
   CIR_PUMP_STP_PB : BOOL ;	//CIRCULATION PUMP STOP PUSH BUTTON
   COOL_FAN_STA_PB : BOOL ;	//COOLER FAN START PUSH BUTTON
   COOL_FAN_STP_PB : BOOL ;	//COOLER FAN STOP PUSH BUTTON
   LAMP_TEST_PB_HYD_LCS : BOOL ;	//LAMP TEST PUSH BUTTON AT HYDRALIC LCS
   ACCUM_STA_PB : BOOL ;	//ACCUMULATOR START PUSH BUTTON
   ACCUM_STP_PB : BOOL ;	//ACCUMULATOR STOP PUSH BUTTON
   SHUTOFF_VALVE_L1_OPEN : BOOL ;	//SHUTOFF VALVE LINE1 OPEN
   SHUTOFF_VALVE_L2_OPEN : BOOL ;	//SHUTOFF VALVE LINE2 OPEN
   LOW_OIL_TEMP : BOOL ;	//LOW OIL TEMPERATURE FROM THERM
   HIGH_OIL_TEMP : BOOL ;	//HIGH OIL TEMPERATURE FROM THERM
   MAXI_OIL_TEMP : BOOL ;	//MAXIMUM OIL TEMPERATURE FROM THERM
   LOW_OIL_LEVEL_FS : BOOL ;	//LOW OIL LEVEL FROM FLOAAT SWITCH
   MIN_OIL_LEVEL_FS : BOOL ;	//MINIMUM OIL LEVEL FROM FLOAAT SWITCH
   RETURN_L1_FILT_CHK : BOOL ;	//RETURN LINE1 FILTER CHOKE
   LOW_OIL_PRESSURE_PS : BOOL ;	//LOW OIL PRESSURE FROM PRESSURE SWITH
   RETURN_L2_FILT_CHK : BOOL ;	//RETURN LINE2 FILTER CHOKE
   HIGH_OIL_PRESSURE_PS : BOOL ;	//HIGH OIL PRESSURE FROM PRESSURE SWITH
   HYD_PUMP1_ON_CMD : BOOL ;	//HYDRALIC PUMP1 ON COMMAND
   HYD_PUMP2_ON_CMD : BOOL ;	//HYDRALIC PUMP2 ON COMMAND
   CIR_PUMP_ON_CMD : BOOL ;	//CIRCULATION PUMP ON COMMAND
   COOL_FAN_ON_CMD : BOOL ;	//COOLER FAN ON COMMAND
   PRE_RELIE_VALVE1_ON_CMD : BOOL ;	//PRESSURE RELIF VALVE1 ON COMMAND
   HYD_SYS_RDY_IND : BOOL ;	//HYDRALIC SYSTEM READY INDICATION
   PUMP1_ON_IND_CD : BOOL ;	//PUMP1 ON INDICATION CD
   PUMP2_ON_IND_CD : BOOL ;	//PUMP2 ON INDICATION CD
   PUMP1_ON_IND_LCS : BOOL ;	//PUMP1 ON INDICATION LCS
   PUMP2_ON_IND_LCS : BOOL ;	//PUMP2 ON INDICATION LCS
   CIRC_PUMP_ON_IND : BOOL ;	//CIRCULATION PUMP ON INDICATION
   COOL_FAN_ON_IND : BOOL ;	//COOLER FAN ON INDICATION
   LOCAL_ON_IND : BOOL ;	//LOCAL ON INDICATION
   HIGH_TEMP_ON_IND : BOOL ;	//HIGH TEMPERATURE ON INDICATION
   LOWER_OIL_LEV_ON_IND : BOOL ;	//LOWER OIL LEVEL ON INDICATION
   FILTER_CHOKE_ON_IND : BOOL ;	//FILTER CHOKE ON INDICATION
   ACCUM_IN_OPE_ON_IND : BOOL ;	//ACCUMULATOR IN OPERATION ON INDICATION
   HEATER_ON_IND : BOOL ;	//HEATER ON INDICATION
   LOW_OIL_TEMP_IND : BOOL ;	//LOW OIL TEMPERATURE INDICATION
   HYDRALI_SYS_HEALTHY : BOOL ;	//HYDRALIC SYSTEM HEALTHY BIT
   HYD_PUMP1_FLT : BOOL ;	//HYDRALIC PUMP1 FAULT
   HYD_FUN_PULSE1 : BOOL ;	//HYDRALIC FUNCTION PULSE1
   HYD_PUMP1_FLT_TMR : INT ;	//HYDRALIC PUMP1 FAULT TIMER
   HYD_PUMP1_FLT_GEN_TIME : INT ;	//HYDRALIC PUMP1 FAULT GENERATION TIME SET
   HYD_PUMP2_FLT : BOOL ;
   HYD_FUN_PULSE2 : BOOL ;
   HYD_FUN_PULSE3 : BOOL ;
   HYD_FUN_PULSE4 : BOOL ;
   HYD_FUN_PULSE5 : BOOL ;
   HYD_FUN_PULSE6 : BOOL ;
   PRE_RELIE_VALVE2_ON_CMD : BOOL ;	//PRESSURE RELIF VALVE2 ON COMMAND
   HYD_PUMP2_FLT_TMR : INT ;	//HYDRALIC PUMP2 FAULT TIMER
   HYD_PUMP2_FLT_GEN_TIME : INT ;	//HYDRALIC PUMP2 FAULT GENERATION TIME SET
   HYD_PRE_RLV_VAL1_TMR : INT ;	//HYDRALIC PRESSURE RELIVE VALVE1 OPEN TIMER
   HYD_PRE_RLV_VAL1_SET_TIM : INT ;	//HYDRALIC PRESSURE RELIVE VALVE1 OPEN SET TIME SET
   HYD_PRE_RLV_VAL2_TMR : INT ;	//HYDRALIC PRESSURE RELIVE VALVE2 OPEN TIMER
   HYD_PRE_RLV_VAL2_SET_TIM : INT ;	//HYDRALIC PRESSURE RELIVE VALVE2 OPEN SET TIME SET
   HYD_SYS_READY_BIT : BOOL ;	//HYDRALIC SYSTEM READY BIT
   HYD_CIR_PUMP_FLT : BOOL ;	//HYDRALIC CIRCULATION PUMP FAULT
   HYD_COOL_FAN_FLT : BOOL ;	//HYDRALIC COOLER FAN FAULT
   EMG_ACC_ON_CMD : BOOL ;	//EMERGENCY ACCUMULATOR ON COMMAND
   HYD_CIR_PUMP_FLT_TMR : INT ;	//HYDRALIC CIRCULATION PUMP FAULT TIMER
   HYD_CIRPUMP_FLT_GEN_TIME : INT ;	//HYDRALIC CIRCULATION PUMP FAULT GENERATION TIME SET
   HYD_COOL_FAN_FLT_TMR : INT ;	//HYDRALIC COOLER FAN FAULT TIMER
   HYD_COOL_FA_FLT_GEN_TIME : INT ;	//HYDRALIC COOLER FAN FAULT GENERATION TIME SET
   PRE_RLV_VLV1_RST_TIME : BOOL ;	//PRESSURE RELIVE VALVE 1 RESET BIT
   PRE_RLV_VLV2_RST_TIME : BOOL ;	//PRESSURE RELIVE VALVE 2 RESET BIT
  END_STRUCT ;	
BEGIN
   HYD_PUMP1_FLT_GEN_TIME := 5;
   HYD_PUMP2_FLT_GEN_TIME := 3;
   HYD_PRE_RLV_VAL1_SET_TIM := 5;
   HYD_PRE_RLV_VAL2_SET_TIM := 5;
   HYD_CIRPUMP_FLT_GEN_TIME := 5;
   HYD_COOL_FA_FLT_GEN_TIME := 5;
END_DATA_BLOCK

DATA_BLOCK "TRAVEL_DRIVE_DB"	// DB 3
VERSION : 0.1
  STRUCT
   TRA_GRP_1_RDY_FOR_STA : BOOL ;	//TRAVEL GROUP1 READY FOR START
   TRA_GRP_1_RUN_FB : BOOL ;	//TRAVEL GROUP1 RUN FEEDBACK
   TRA_MOTOR_1_OLR : BOOL ;	//TRAVEL MOTOR1 OLR
   TRA_MOTOR_2_OLR : BOOL ;	//TRAVEL MOTOR2 OLR
   SIREN_RDY_FOR_STA : BOOL ;	//SIREN READY FOR START
   SIREN_RUN_FB : BOOL ;	//SIREN RUNING FEEDBACK
   HOPPER_STOP_PB : BOOL ;	//HOPPER STOP PUSHBUTTON
   SIREN_OLR_TRIP : BOOL ;	//SIREN OVER LOAD TRIP
   BRAKE_1_RDY_FOR_STA : BOOL ;	//BRAKE1 READY FOR START
   BRAKE_1_RUN_FB : BOOL ;	//BRAKE1 RUN FEEDBACK
   TRA_GRP_2_RDY_FOR_STA : BOOL ;	//TRAVEL GROUP2 READY FOR START
   TRA_GRP_2_RUN_FB : BOOL ;	//TRAVEL GROUP2 RUN FEEDBACK
   TRA_MOTOR_3_OLR : BOOL ;	//TRAVEL MOTOR3 OLR
   TRA_MOTOR_4_OLR : BOOL ;	//TRAVEL MOTOR4 OLR
   BRAKE_2_RDY_FOR_STA : BOOL ;	//BRAKE2 READY FOR START
   BRAKE_2_RUN_FB : BOOL ;	//BRAKE2 RUN FEEDBACK
   TRA_JS_HOME_PB : BOOL ;	//TRAVEL JOYSTICK HOME PUSHBUTTON
   TRA_JS_FWD_PB : BOOL ;	//TRAVEL JOYSTICK FORWARD PUSHBUTTON
   TRA_JS_REV_PB : BOOL ;	//TRAVEL JOYSTICK REVERSE PUSHBUTTON
   TRA_DEAD_MAN_BUTTON : BOOL ;	//TRAVEL DEADMAN BUTTON
   LASER_SPOTTING : BOOL ;	//LASER SPOTTING
   DRIVE1_HW_PROFI_SS : BOOL ;	//DRIVE1 HARDWARE OR PROFIBUS SELECTOR SWITCH
   DRIVE1_RUN_FB : BOOL ;	//DRIVE1 RUN FEEDBACK
   DRIVE_1_RDY_FOR_STA : BOOL ;	//DRIVE1 READY FOR START
   DRIVE1_TRIP_FB : BOOL ;	//DRIVE1 TRIP FEEDBACK
   DRIVE2_HW_PROFI_SS : BOOL ;	//DRIVE2 HARDWARE OR PROFIBUS SELECTOR SWITCH
   DRIVE2_RUN_FB : BOOL ;	//DRIVE2 RUN FEEDBACK
   DRIVE_2_RDY_FOR_STA : BOOL ;	//DRIVE2 READY FOR START
   DRIVE2_TRIP_FB : BOOL ;	//DRIVE2 TRIP FEEDBACK
   LS_END_FWD_FB : BOOL ;	//LIMIT SWITCH END FORWARD FEEDBACK
   LONG_TRA_SLOW_SPD : BOOL ;	//LONG TRAVEL SLOW SPEED
   LS_END_REV_FB : BOOL ;	//LIMIT SWITCH END REVERSE FEEDBACK
   TRA_GRP1_ON_CMD : BOOL ;	//TRAVEL GROUP1 ON COMMAND
   TRA_GRP2_ON_CMD : BOOL ;	//TRAVEL GROUP2 ON COMMAND
   SIREN_ON_CMD : BOOL ;	//SIREN ON COMMAND
   BRAKE1_ON_CMD : BOOL ;	//BRAKE1 ON COMMAND
   BRAKE2_ON_CMD : BOOL ;	//BRAKE2 ON COMMAND
   AUDIO_VIS_ALRM_ON_CMD : BOOL ;	//AUDIO VISUAL ALARAM ON COMMAND
   TRA_DRIVE_FWD : BOOL ;	//TRAVEL DRIVE FORWARD
   TRA_DRIVE_REV : BOOL ;	//TRAVEL DRIVE REVERSE
   LOG_INPUT_1_TRA_DRIVE : BOOL ;	//LOGIC INPUT1 TO TRAVEL DRIVE
   LOG_INPUT_2_TRA_DRIVE : BOOL ;	//LOGIC INPUT2 TO TRAVEL DRIVE
   LOG_INPUT_3_TRA_DRIVE : BOOL ;	//LOGIC INPUT3 TO TRAVEL DRIVE
   TRA_PERMISSION_IND : BOOL ;	//TRAVEL PERMISSION INDICATION
   TRA_D1_FWD_ON_CMD : BOOL ;	//TRAVEL DRIVE1 FORWARD ON COMMAND
   TRA_D1_REV_ON_CMD : BOOL ;	//TRAVEL DRIVE1 REVERSE ON COMMAND
   TRA_D2_FWD_ON_CMD : BOOL ;	//TRAVEL DRIVE2 FORWARD ON COMMAND
   TRA_D2_REV_ON_CMD : BOOL ;	//TRAVEL DRIVE2 REVERSE ON COMMAND
   TRA_AUTO_MAN_SS : BOOL ;	//TRAVEL AUTO OR MANUAL SELECTOR SWITCH
   TRA_INT_LOCK_BIT : BOOL ;	//TRAVEL OPERATION INTERLOCK BIT
   TRA_FWD_CHANGE_OVER_DELA : BOOL ;	//TRAVEL DRIVE FORWARD CHANGE OVER DELAY
   TRA_PULSE_1 : BOOL ;
   TRA_PULSE_2 : BOOL ;
   TRA_PULSE_3 : BOOL ;
   TRA_PULSE_4 : BOOL ;
   TRA_PULSE_5 : BOOL ;
   SPARE_1 : INT ;
   SPARE_2 : INT ;
   SPARE_3 : INT ;
   SPARE_4 : INT ;
   SPARE_5 : INT ;
   SPARE_6 : INT ;
   SPARE_7 : INT ;
   SPARE_8 : INT ;
   TRA_FWD_1_FB_FLT : BOOL ;
   TRA_FWD_2_FB_FLT : BOOL ;
   TRA_REV_1_FB_FLT : BOOL ;
   TRA_REV_2_FB_FLT : BOOL ;
   TRA_REV_CHANGE_OVER_DELA : BOOL ;	//TRAVEL DRIVE REVERSE CHANGE OVER DELAY
   TRA_BRAKE_1_2_FAULT : BOOL ;	//TRAVEL GROUP BRAKE 1 & BRAKE 2 FAULT
   TRA_AUTO_POS_ACK_SET : BOOL ;	//TRAVEL AUTO POSITION ACKNOWLEDGE SET BIT
   TRA_GRP_BR_FAULT_GEN_TMR : INT ;	//TRAVEL GROUP BRAKE FAULT GENERATION TIMER
   TRA_GRP_BR_FAULT_GEN_TIM : INT ;	//TRAVEL GROUP BRAKE FAULT GENERATION TIME SET
   TRA_SPEED_REF_FROM_JS : INT ;	//TRAVEL SPEED REFERNCE FROM JOY STICK
   TRA_JS_REF_NEG_REM : INT ;	//TRAVEL JOY STICK NEGEATIVE SPEED REFERENCE REMOVED
   TRA_JS_INT_TO_DI : DINT ;	//TRAVEL JOY STICK INTEGER TO DOUBLE INTEGER
   TRA_JS_DI_TO_REAL : REAL ;	//TRAVEL JOY STICK   DOUBLE INTEGER TO REAL
   TRA_JS_UN_SCA_RET_VAL : WORD ;	//TRAVEL JOY STICK UNSCALE RETURN VALUE
   TRA_SPEED_REF_VALUE : INT ;	//TRAVEL SPEED REFERENCE VALUE
   TRA_D1_FWD_ON_CMD_PF : BOOL ;	//TRAVEL DRIVE1 FORWARD ON COMMAND IN PROFIBUS
   TRA_D1_REV_ON_CMD_PF : BOOL ;	//TRAVEL DRIVE1 REVERSE ON COMMAND IN PROFIBUS
   TRA_D2_FWD_ON_CMD_PF : BOOL ;	//TRAVEL DRIVE2 FORWARD ON COMMAND IN PROFIBUS
   TRA_D2_REV_ON_CMD_PF : BOOL ;	//TRAVEL DRIVE2 REVERSE ON COMMAND IN PROFIBUS
   TRAVEL_PF_BUS_SPARE : BOOL ;	//TRAVEL PROFIBUS SPARE
   TRAVEL_PF_BUS_SPARE1 : BOOL ;	//TRAVEL PROFIBUS SPARE
   TRAVEL_PF_BUS_SPARE2 : BOOL ;	//TRAVEL PROFIBUS SPARE
   TRAVEL_PF_BUS_SPARE3 : BOOL ;	//TRAVEL PROFIBUS SPARE
   TRA_JS_INT_TO_DI_PF : DINT ;	//TRAVEL JOY STICK INTEGER TO DOUBLE INTEGER PROFIBUS
   TRA_JS_DI_TO_REAL_PF : REAL ;	//TRAVEL JOY STICK   DOUBLE INTEGER TO REAL PROFIBUS
   TRA_SPEED_REF_VALUE_PF : INT ;	//TRAVEL SPEED REFERENCE VALUE PROFIBUS
   TRA_INTER_BYPASS : BOOL ;	//TRAVEL INTERLOCK BYPASS
   TRA_INTERLOCK_1 : BOOL ;	//TRAVEL INTERLOCK
   LT_HOOT_SIR_PB : BOOL ;	//LONG TRAVEL HOOTER PUSH BUTTON
   LT_HOOT_SIR_CMD : BOOL ;	//LONG TRAVEL HOOTER COMMAND
  END_STRUCT ;	
BEGIN
   TRA_GRP_BR_FAULT_GEN_TIM := 5;
END_DATA_BLOCK

DATA_BLOCK "CC_BUNKER_GATE_DB"	// DB 4
VERSION : 0.1
  STRUCT
   BUNKER_GATE : STRUCT
    MAN_MD : BOOL ;	//BUNKER GATE MANUAL MODE
    REP_MD : BOOL ;	//BUNKER GATE REPAIR MODE
    SA_MD : BOOL ;	//BUNKER GATE SEMI AUTO MODE
    BG_1_UP_STA_PB : BOOL ;	//BUNKER GATE 1 UP START PUSH BUTTON
    BG_1_DN_STA_PB : BOOL ;	//BUNKER GATE 1 DOWN START PUSH BUTTON
    BG_1_HM_STA_PB : BOOL ;	//BUNKER GATE 1 HOME START PUSH BUTTON
    BG_1_OPN_STA_PB : BOOL ;	//BUNKER GATE 1 OPEN START PUSH BUTTON
    BG_1_CLS_STA_PB : BOOL ;	//BUNKER GATE 1 CLOSE START PUSH BUTTON
    BG_2_UP_STA_PB : BOOL ;	//BUNKER GATE 2 UP START PUSH BUTTON
    BG_2_DN_STA_PB : BOOL ;	//BUNKER GATE 2 DOWN START PUSH BUTTON
    BG_2_HM_STA_PB : BOOL ;	//BUNKER GATE 2 HOME START PUSH BUTTON
    BG_2_OPN_STA_PB : BOOL ;	//BUNKER GATE 2 OPEN START PUSH BUTTON
    BG_2_CLS_STA_PB : BOOL ;	//BUNKER GATE 2 CLOSE START PUSH BUTTON
    BG_3_UP_STA_PB : BOOL ;	//BUNKER GATE 3 UP START PUSH BUTTON
    BG_3_DN_STA_PB : BOOL ;	//BUNKER GATE 3 DOWN START PUSH BUTTON
    BG_3_HM_STA_PB : BOOL ;	//BUNKER GATE 3 HOME START PUSH BUTTON
    BG_3_OPN_STA_PB : BOOL ;	//BUNKER GATE 3 OPEN START PUSH BUTTON
    BG_3_CLS_STA_PB : BOOL ;	//BUNKER GATE 3 CLOSE START PUSH BUTTON
    COAL_LD_STA_PB : BOOL ;	//BUNKER GATE COAL LOAD START PUSH BUTTON
    COAL_LD_STP_PB : BOOL ;	//BUNKER GATE COAL LOAD STOP PUSH BUTTON
    BG_1_UP_LS : BOOL ;	//BUNKER GATE 1 UP LIMIT SWITCH
    BG_1_DN_LS : BOOL ;	//BUNKER GATE 1 DOWN LIMIT SWITCH
    BG_1_HM_LS : BOOL ;	//BUNKER GATE 1 HOME LIMIT SWITCH
    BG_1_OPN_LS : BOOL ;	//BUNKER GATE 1 OPEN LIMIT SWITCH
    BG_1_CLS_LS : BOOL ;	//BUNKER GATE 2 CLOSE LIMIT SWITCH
    BG_2_UP_LS : BOOL ;	//BUNKER GATE 2 UP LIMIT SWITCH
    BG_2_DN_LS : BOOL ;	//BUNKER GATE 2 DOWN LIMIT SWITCH
    BG_2_HM_LS : BOOL ;	//BUNKER GATE 2 HOME LIMIT SWITCH
    BG_2_OPN_LS : BOOL ;	//BUNKER GATE 2 OPEN LIMIT SWITCH
    BG_2_CLS_LS : BOOL ;	//BUNKER GATE 2 CLOSE LIMIT SWITCH
    BG_3_UP_LS : BOOL ;	//BUNKER GATE 3 UP LIMIT SWITCH
    BG_3_DN_LS : BOOL ;	//BUNKER GATE 3 DOWN LIMIT SWITCH
    BG_3_HM_LS : BOOL ;	//BUNKER GATE 3 HOME LIMIT SWITCH
    BG_3_OPN_LS : BOOL ;	//BUNKER GATE 3 OPEN LIMIT SWITCH
    BG_3_CLS_LS : BOOL ;	//BUNKER GATE 3 CLOSE LIMIT SWITCH
    HOP_1_MAX_LS : BOOL ;	//HOPPER 1 MAXIMUM LIMIT SWITCH
    HOP_2_MAX_LS : BOOL ;	//HOPPER 2 MAXIMUM LIMIT SWITCH
    HOP_3_MAX_LS : BOOL ;	//HOPPER 3 MAXIMUM LIMIT SWITCH
    BG_1_UP_STA_PB_LCS : BOOL ;	//BUNKER GATE 1 UP LOCAL START PUSH BUTTON
    BG_1_DN_STA_PB_LCS : BOOL ;	//BUNKER GATE 1 DOWN LOCAL START PUSH BUTTON
    BG_1_HM_STA_PB_LCS : BOOL ;	//BUNKER GATE 1 HOME LOCAL START PUSH BUTTON
    BG_1_OPN_STA_PB_LCS : BOOL ;	//BUNKER GATE 1 OPEN LOCAL START PUSH BUTTON
    BG_1_CLS_STA_PB_LCS : BOOL ;	//BUNKER GATE 1 CLOSE LOCAL START PUSH BUTTON
    BG_2_UP_STA_PB_LCS : BOOL ;	//BUNKER GATE 2 UP START LOCAL PUSH BUTTON
    BG_2_DN_STA_PB_LCS : BOOL ;	//BUNKER GATE 2 DOWN LOCAL START PUSH BUTTON
    BG_2_HM_STA_PB_LCS : BOOL ;	//BUNKER GATE 2 HOME LOCAL START PUSH BUTTON
    BG_2_OPN_STA_PB_LCS : BOOL ;	//BUNKER GATE 2 OPEN LOCAL START PUSH BUTTON
    BG_2_CLS_STA_PB_LCS : BOOL ;	//BUNKER GATE 2 CLOSE LOCAL START PUSH BUTTON
    BG_3_UP_STA_PB_LCS : BOOL ;	//BUNKER GATE 3 UP LOCAL START PUSH BUTTON
    BG_3_DN_STA_PB_LCS : BOOL ;	//BUNKER GATE 3 DOWN LOCAL START PUSH BUTTON
    BG_3_OPN_STA_PB_LCS : BOOL ;	//BUNKER GATE 3 OPEN LOCAL START PUSH BUTTON
    BG_3_CLS_STA_PB_LCS : BOOL ;	//BUNKER GATE 3 CLOSE LOCAL START PUSH BUTTON
    BG_1_UP_CMD : BOOL ;	//BUNKER GATE 1 UP COMMAND
    BG_1_DN_CMD : BOOL ;	//BUNKER GATE 1 DOWN COMMAND
    BG_1_OPN_CMD : BOOL ;	//BUNKER GATE 1 OPEN COMMAND
    BG_1_CLS_CMD : BOOL ;	//BUNKER GATE 1 CLOSE COMMAND
    BG_2_UP_CMD : BOOL ;	//BUNKER GATE 2 UP COMMAND
    BG_2_DN_CMD : BOOL ;	//BUNKER GATE 2 DOWN COMMAND
    BG_2_OPN_CMD : BOOL ;	//BUNKER GATE 2 OPEN COMMAND
    BG_2_CLS_CMD : BOOL ;	//BUNKER GATE 2 CLOSE COMMAND
    BG_3_UP_CMD : BOOL ;	//BUNKER GATE 3 UP COMMAND
    BG_3_DN_CMD : BOOL ;	//BUNKER GATE 3 DOWN COMMAND
    BG_3_OPN_CMD : BOOL ;	//BUNKER GATE 3 OPEN COMMAND
    BG_3_CLS_CMD : BOOL ;	//BUNKER GATE 3 CLOSE COMMAND
    BG_1_UP_IND : BOOL ;	//BUNKER GATE 1 UP INDICATION
    BG_1_DN_IND : BOOL ;	//BUNKER GATE 1 DOWN INDICATION
    BG_1_OPN_IND : BOOL ;	//BUNKER GATE 1 OPEN INDICATION
    BG_1_CLS_IND : BOOL ;	//BUNKER GATE 1 CLOSE INDICATION
    BG_1_HME_IND : BOOL ;	//BUNKER GATE 1 HOME INDICATION
    BG_1_UP_IND_LCS : BOOL ;	//BUNKER GATE 1 UP INDICATION LCS
    BG_1_DN_IND_LCS : BOOL ;	//BUNKER GATE 1 DOWN INDICATION LCS
    BG_1_OPN_IND_LCS : BOOL ;	//BUNKER GATE 1 OPEN INDICATION LCS
    BG_1_CLS_IND_LCS : BOOL ;	//BUNKER GATE 1 CLOSE INDICATION LCS
    BG_1_HME_IND_LCS : BOOL ;	//BUNKER GATE 1 HOME INDICATION LCS
    BG_2_UP_IND : BOOL ;	//BUNKER GATE 2 UP INDICATION
    BG_2_DN_IND : BOOL ;	//BUNKER GATE 2 DOWN INDICATION
    BG_2_OPN_IND : BOOL ;	//BUNKER GATE 2 OPEN INDICATION
    BG_2_CLS_IND : BOOL ;	//BUNKER GATE 2 CLOSE INDICATION
    BG_2_HME_IND : BOOL ;	//BUNKER GATE 2 HOME INDICATION
    BG_2_UP_IND_LCS : BOOL ;	//BUNKER GATE 2 UP INDICATION LCS
    BG_2_DN_IND_LCS : BOOL ;	//BUNKER GATE 2 DOWN INDICATION LCS
    BG_2_OPN_IND_LCS : BOOL ;	//BUNKER GATE 2 OPEN INDICATION LCS
    BG_2_CLS_IND_LCS : BOOL ;	//BUNKER GATE 2 CLOSE INDICATION LCS
    BG_2_HME_IND_LCS : BOOL ;	//BUNKER GATE 2 HOME INDICATION LCS
    BG_3_UP_IND : BOOL ;	//BUNKER GATE 3 UP INDICATION
    BG_3_DN_IND : BOOL ;	//BUNKER GATE 3 DOWN INDICATION
    BG_3_OPN_IND : BOOL ;	//BUNKER GATE 3 OPEN INDICATION
    BG_3_CLS_IND : BOOL ;	//BUNKER GATE 3 CLOSE INDICATION
    BG_3_HME_IND : BOOL ;	//BUNKER GATE 3 HOME INDICATION
    BG_3_UP_IND_LCS : BOOL ;	//BUNKER GATE 3 UP INDICATION LCS
    BG_3_DN_IND_LCS : BOOL ;	//BUNKER GATE 3 DOWN INDICATION LCS
    BG_3_OPN_IND_LCS : BOOL ;	//BUNKER GATE 3 OPEN INDICATION LCS
    BG_3_CLS_IND_LCS : BOOL ;	//BUNKER GATE 3 CLOSE INDICATION LCS
    BG_3_HME_IND_LCS : BOOL ;	//BUNKER GATE 3 HOME INDICATION LCS
    HOP_1_MAX_IND : BOOL ;	//HOPPER 1 MAXIMUM INDICATION
    HOP_2_MAX_IND : BOOL ;	//HOPPER 2 MAXIMUM INDICATION
    HOP_3_MAX_IND : BOOL ;	//HOPPER 3 MAXIMUM INDICATION
    BG_COAL_LD_IND : BOOL ;	//BUNKER COAL LOAD INDICATION
    BG_COAL_LD_PROG_IND : BOOL ;	//BUNKER COAL LOADING PROGRESS INDICATION
    INTERLOCK_BIT : BOOL ;	//BUNKER GATE INTERLOCK BIT
    LCS_MD : BOOL ;	//BUNKER GATE LCS MODE
    COAL_LD_STA_PB_AUTO_SET : BOOL ;	//COAL LOADING START PUSH BUTTON AUTO SEQUENCE SET BIT
    COAL_LD_STP_PB_AUTO_SET : BOOL ;	//COAL LOADING STOP PUSH BUTTON AUTO SEQUENCE SET BIT
    PULSE_1 : BOOL ;
    PULSE_2 : BOOL ;
    PULSE_3 : BOOL ;
    PULSE_4 : BOOL ;
    PULSE_5 : BOOL ;
    PULSE_6 : BOOL ;
    PULSE_7 : BOOL ;
    PULSE_8 : BOOL ;
    PULSE_9 : BOOL ;
    BG_1_AUTO_UP_CMD_RCHD : BOOL ;	//BUNKER GATE 1 AUTO UP COMMAND REACHED
    BG_1_AUTO_OPN_CMD_RCHD : BOOL ;	//BUNKER GATE 1 AUTO OPEN COMMAND REACHED
    BG_1_AUTO_CLS_CMD_RCHD : BOOL ;	//BUNKER GATE 1 AUTO CLOSE COMMAND REACHED
    BG_1_AUTO_OPN_RCHD_HME : BOOL ;	//BUNKER GATE 1 AUTO OPEN COMMAND REACHED WITH HOPPER MAXIMUM
    BG_1_AUTO_DN_CMD_RCHD : BOOL ;	//BUNKER GATE 1 AUTO DOWN COMMAND REACHED
    BG_2_AUTO_UP_CMD_RCHD : BOOL ;	//BUNKER GATE 2 AUTO UP COMMAND REACHED
    BG_2_AUTO_OPN_CMD_RCHD : BOOL ;	//BUNKER GATE 2 AUTO OPEN COMMAND REACHED
    BG_2_AUTO_CLS_CMD_RCHD : BOOL ;	//BUNKER GATE 2 AUTO CLOSE COMMAND REACHED
    BG_2_AUTO_OPN_RCHD_HME : BOOL ;	//BUNKER GATE 2 AUTO OPEN COMMAND REACHED WITH HOPPER MAXIMUM
    BG_2_AUTO_DN_CMD_RCHD : BOOL ;	//BUNKER GATE 2 AUTO DOWN COMMAND REACHED
    BG_3_AUTO_UP_CMD_RCHD : BOOL ;	//BUNKER GATE 3 AUTO UP COMMAND REACHED
    BG_3_AUTO_OPN_CMD_RCHD : BOOL ;	//BUNKER GATE 3 AUTO OPEN COMMAND REACHED
    BG_3_AUTO_CLS_CMD_RCHD : BOOL ;	//BUNKER GATE 3 AUTO CLOSE COMMAND REACHED
    BG_3_AUTO_OPN_RCHD_HME : BOOL ;	//BUNKER GATE 3 AUTO OPEN COMMAND REACHED WITH HOPPER MAXIMUM
    BG_3_AUTO_DN_CMD_RCHD : BOOL ;	//BUNKER GATE 3 AUTO DOWN COMMAND REACHED
    PULSE_10 : BOOL ;
    PULSE_11 : BOOL ;
    PULSE_12 : BOOL ;
    PULSE_13 : BOOL ;
    PULSE_14 : BOOL ;
    PULSE_15 : BOOL ;
    PULSE_16 : BOOL ;
    PULSE_17 : BOOL ;
    PULSE_18 : BOOL ;
    PULSE_19 : BOOL ;
    PULSE_20 : BOOL ;
    PULSE_21 : BOOL ;
    PULSE_22 : BOOL ;
    PULSE_23 : BOOL ;
    PULSE_24 : BOOL ;
    PULSE_25 : BOOL ;
    BG_3_HM_STA_PB_LCS : BOOL ;	//BUNKER GATE HOME START PUSH BUTTON
    BG_LOCAL_IND : BOOL ;	//BUNKER GATE LOCAL INDICATION LCS 91
    BG_LAMP_TEST_PB_LCS_91 : BOOL ;	//BUNKER GATE LAMP TEST PUSH BUTTON LCS 91
    BG_1_HME_CMD : BOOL ;	//BUNKER GATE 1 HOME COMMAND
    BG_2_HME_CMD : BOOL ;	//BUNKER GATE 2 HOME COMMAND
    BG_3_HME_CMD : BOOL ;	//BUNKER GATE 3 HOME COMMAND
    BG_1_HME_OPN_CMD : BOOL ;	//BUNKER GATE 1 HOME AND OPEN COMMAND
    BG_2_HME_OPN_CMD : BOOL ;	//BUNKER GATE 2 HOME AND OPEN COMMAND
    BG_3_HME_OPN_CMD : BOOL ;	//BUNKER GATE 3 HOME AND OPEN COMMAND
    BG_MAN_MODE_CD_LCS : BOOL ;
   END_STRUCT ;
  END_STRUCT ;	
BEGIN
END_DATA_BLOCK

DATA_BLOCK "OVEN_CHARGING_DB"	// DB 5
VERSION : 0.1
  STRUCT
   SF_1_HW_PF_SS : BOOL ;	//SCREW FEEDER 1 HARDWARE/PROFIBUS SELECTOR
   SF_1_RDY_FOR_STA : BOOL ;	//SCREW FEEDER 1 READY FOR START
   SF_1_RUN_FB : BOOL ;	//SCREW FEEDER 1 READY FOR START
   SF_1_TRIP_FB : BOOL ;	//SCREW FEEDER 1 TRIP FEEDBACK
   SF_2_HW_PF_SS : BOOL ;	//SCREW FEEDER 2 HARDWARE/PROFIBUS SELECTOR
   SF_2_RDY_FOR_STA : BOOL ;	//SCREW FEEDER 2 READY FOR START
   SF_2_RUN_FB : BOOL ;	//SCREW FEEDER 2 READY FOR START
   SF_2_TRIP_FB : BOOL ;	//SCREW FEEDER 2 TRIP FEEDBACK
   SF_3_HW_PF_SS : BOOL ;	//SCREW FEEDER 3 HARDWARE/PROFIBUS SELECTOR
   SF_3_RDY_FOR_STA : BOOL ;	//SCREW FEEDER 3 READY FOR START
   SF_3_RUN_FB : BOOL ;	//SCREW FEEDER 3 READY FOR START
   SF_3_TRIP_FB : BOOL ;	//SCREW FEEDER 3 TRIP FEEDBACK
   DC_PWR_PACK : BOOL ;	//DC POWER PACK
   SF_1_STA_PB : BOOL ;	//SCREW FEEDER 1 START PUSH BUTTON
   SF_1_STP_PB : BOOL ;	//SCREW FEEDER 1 STOP PUSH BUTTON
   SF_1_HI_SEL : BOOL ;	//SCREW FEEDER 1 HIGH SPEED SELECT
   SF_1_LO_SEL : BOOL ;	//SCREW FEEDER 1 LOW SPEED SELECT
   SF_2_STA_PB : BOOL ;	//SCREW FEEDER 2 START PUSH BUTTON
   SF_2_STP_PB : BOOL ;	//SCREW FEEDER 2 STOP PUSH BUTTON
   SF_2_HI_SEL : BOOL ;	//SCREW FEEDER 2 HIGH SPEED SELECT
   SF_2_LO_SEL : BOOL ;	//SCREW FEEDER 2 LOW SPEED SELECT
   SF_3_STA_PB : BOOL ;	//SCREW FEEDER 3 START PUSH BUTTON
   SF_3_STP_PB : BOOL ;	//SCREW FEEDER 3 STOP PUSH BUTTON
   SF_3_HI_SEL : BOOL ;	//SCREW FEEDER 3 HIGH SPEED SELECT
   SF_3_LO_SEL : BOOL ;	//SCREW FEEDER 3 LOW SPEED SELECT
   SL_GT_1_CLS_STA_PB : BOOL ;	//SLIDE GATE 1 CLOSE START PUSH BUTTON
   SL_GT_1_OPN_STA_PB : BOOL ;	//SLIDE GATE 1 OPEN START PUSH BUTTON
   SL_GT_2_CLS_STA_PB : BOOL ;	//SLIDE GATE 2 CLOSE START PUSH BUTTON
   SL_GT_2_OPN_STA_PB : BOOL ;	//SLIDE GATE 2 OPEN START PUSH BUTTON
   SL_GT_3_CLS_STA_PB : BOOL ;	//SLIDE GATE 3 CLOSE START PUSH BUTTON
   SL_GT_3_OPN_STA_PB : BOOL ;	//SLIDE GATE 3 OPEN START PUSH BUTTON
   SL_GT_1_CLS_LS : BOOL ;	//SLIDE GATE 1 CLOSE LIMIT SWITCH (FWD LS)
   SL_GT_1_OPN_LS : BOOL ;	//SLIDE GATE 1 OPEN LIMIT SWITCH (REV LS)
   SL_GT_2_CLS_LS : BOOL ;	//SLIDE GATE 2 CLOSE LIMIT SWITCH (FWD LS)
   SL_GT_2_OPN_LS : BOOL ;	//SLIDE GATE 2 OPEN LIMIT SWITCH (REV LS)
   SL_GT_3_CLS_LS : BOOL ;	//SLIDE GATE 3 CLOSE LIMIT SWITCH (FWD LS)
   SL_GT_3_OPN_LS : BOOL ;	//SLIDE GATE 3 OPEN LIMIT SWITCH (REV LS)
   OVEN_CHARGING_PB : BOOL ;	//OVEN CHARGING AUTO START PUSHBUTTON
   FINISH_CHR_PB : BOOL ;	//FINISH CHARGING PUSH BUTTON
   INPUT_SPARE2 : BOOL ;	//INPUT SPARE
   SF1_HIGH_SPEED_CMD : BOOL ;	//SCREW FEEDER 1 HIGH SPEED COMMAND
   SF1_LOW_SPEED_CMD : BOOL ;	//SCREW FEEDER 1 LOW SPEED COMMAND
   SF2_HIGH_SPEED_CMD : BOOL ;	//SCREW FEEDER 2 HIGH SPEED COMMAND
   SF2_LOW_SPEED_CMD : BOOL ;	//SCREW FEEDER 2 LOW SPEED COMMAND
   SF3_HIGH_SPEED_CMD : BOOL ;	//SCREW FEEDER 3 HIGH SPEED COMMAND
   SF3_LOW_SPEED_CMD : BOOL ;	//SCREW FEEDER 3 LOW SPEED COMMAND
   SF1_ON_IND : BOOL ;	//SCREW FEEDER 1 ON INDICATION
   SF2_ON_IND : BOOL ;	//SCREW FEEDER 2 ON INDICATION
   SF3_ON_IND : BOOL ;	//SCREW FEEDER 3 ON INDICATION
   SL_GT_1_CLS_CMD : BOOL ;	//SLIDE GATE 1 CLOSE COMMAND
   SL_GT_1_OPN_CMD : BOOL ;	//SLIDE GATE 1 OPEN COMMAND
   SL_GT_1_CLS_IND : BOOL ;	//SLIDE GATE 1 CLOSE INDICATION
   SL_GT_1_OPN_IND : BOOL ;	//SLIDE GATE 1 OPEN INDICAATION
   SL_GT_2_CLS_CMD : BOOL ;	//SLIDE GATE 2 CLOSE COMMAND
   SL_GT_2_OPN_CMD : BOOL ;	//SLIDE GATE 2 OPEN COMMAND
   SL_GT_2_CLS_IND : BOOL ;	//SLIDE GATE 2 CLOSE INDICATION
   SL_GT_2_OPN_IND : BOOL ;	//SLIDE GATE 2 OPEN INDICAATION
   SL_GT_3_CLS_CMD : BOOL ;	//SLIDE GATE 3 CLOSE COMMAND
   SL_GT_3_OPN_CMD : BOOL ;	//SLIDE GATE 3 OPEN COMMAND
   SL_GT_3_CLS_IND : BOOL ;	//SLIDE GATE 3 CLOSE INDICATION
   SL_GT_3_OPN_IND : BOOL ;	//SLIDE GATE 3 OPEN INDICAATION
   CHR_PER_IND : BOOL ;	//CHARGING PERMISSION INDICATION
   CHR_CMP_IND : BOOL ;	//CHARGING COMPLETED INDICATION
   PREP_CHR_IND : BOOL ;	//PREPEARE TO CHARGE INDICATION
   OVEN_CHR_IND : BOOL ;	//OVEN CHARGING IND
   FNSH_CHR_IND : BOOL ;	//FINISH CHARGING INDICATION
   OUTPUT_SPARE : BOOL ;	//OUTPUT SPARE
   OUTPUT_SPARE1 : BOOL ;	//OUTPUT SPARE
   OUTPUT_SPARE2 : BOOL ;	//OUTPUT SPARE
   OUTPUT_SPARE3 : BOOL ;	//OUTPUT SPARE
   OUTPUT_SPARE4 : BOOL ;	//OUTPUT SPARE
   LID_START_OVEN_CHR_LOW : BOOL ;	//LID AUTO START OVEN CHARGE IN LOW SPEED
   OVEN_CHR_INTR_BIT : BOOL ;	//OVEN CHARGE INTERLOCK SATISFIED BIT
   OVEN_CHR_AUTO_MODE : BOOL ;	//OVEN CHARGE AUTO MODE SS
   OVEN_CHR_MANUAL_MODE : BOOL ;	//OVEN CHARGE MANUAL MODE SS
   OVEN_CHR_REPARE_MODE : BOOL ;	//OVEN CHARGE REPARE MODE SS
   SL_GT_1_OP_CUT : BOOL ;	//SLIDE GATE OPEN OPERATION COMPLETED BIT
   SL_GT_1_CLS_CUT : BOOL ;	//SLIDE GATE CLOSE OPERATION COMPLETED BIT
   SF1_MOTOR_FLT_BIT : BOOL ;	//SCREW FEEDER MOTOR 1 FAULT GENERATED
   SL_GT_1_PULSE : BOOL ;	//SLIDE GATE 1 PULSE
   SL_GT_1_OP_TMR : INT ;	//SLIDE GATE OPEN OPERATION COMPLETED TIMER
   SL_GT_1_OP_TIME : INT ;	//SLIDE GATE OPEN OPERATION COMPLETED TIME
   SL_GT_1_CLS_TMR : INT ;	//SLIDE GATE CLOSE OPERATION COMPLETED TIMER
   SL_GT_1_CLS_TIME : INT ;	//SLIDE GATE CLOSE OPERATION COMPLETED TIME
   SF1_FLT_OP_TMR : INT ;	//SCREW FEEDER 1 FAULT OPERATED TIMER
   SF1_FLT_OP_TIME : INT ;	//SCREW FEEDER 1 FAULT OPERATED TIME
   SF1_ENC_PER_REV : DINT ;	//SCREW FEEDER 1 ENCODER PER REVOLUTION
   SF1_HIGH_SPD_COUNT_SET : DINT ;	//SCREW FEEDER 1 HIGH SPEED SET POINT
   SF1_LOW_SPD_COUNT_SET : DINT ;	//SCREW FEEDER 1 LOW SPEED SET POINT
   SF1_HI_SPD_CNT_OVER_BIT : BOOL ;	//SCREW FEEDER 1 HIGH SPEED COUNT OVER
   SF1_LO_SPD_CNT_OVER_BIT : BOOL ;	//SCREW FEEDER 1 LOW SPEED COUNT OVER
   SF1_RST_FOR_LOW_SPD_STA : BOOL ;	//SCREW FEEDER 1 RESET FOR LOW SPEED START
   LID_START_OVEN_CHR_HI : BOOL ;	//LID AUTO START OVEN CHARGE IN HIGH SPEED
   SL_GT_1_PULSE1 : BOOL ;	//SLIDE GATE 1 PULSE
   SF1_PULSE : BOOL ;	//SCREW FEEDER 1 PULSE
   SL_GT_1_PULSE2 : BOOL ;	//SLIDE GATE 1 PULSE
   OVEN_CHR_SF1_HI_SPD_STA : BOOL ;	//SCREW FEEDER 1 HIGH SPEED SET IN AUTO
   SF1_ENCODE_PROXI_MODE : BOOL ;	//SCREW FEEDER 1 PROXIMITY MODE SELECTION
   SF2_ENCODE_PROXI_MODE : BOOL ;	//SCREW FEEDER 2 PROXIMITY MODE SELECTION
   SF3_ENCODE_PROXI_MODE : BOOL ;	//SCREW FEEDER 3 PROXIMITY MODE SELECTION
   SF1_PROXI_PULSE : BOOL ;	//SCREW FEEDER 1 PROXIMITY INPUT PULSE
   SF1_HIGH_SPEED_CMD_PF : BOOL ;	//SCREW FEEDER 1 HIGH SPEED COMMAND PROFIBUS
   SF1_LOW_SPEED_CMD_PF : BOOL ;	//SCREW FEEDER 1 LOW SPEED COMMAND PROFIBUS
   SF1_PULSE_20 : BOOL ;	//SCREW FEEDER 1 PULSE USED IN NETWORK 11
   SF1_PULSE_21 : BOOL ;	//SCREW FEEDER 1 PULSE USED IN NETWORK 12
   SF1_SPARE_MEMORY_WORD : WORD ;
   SF1_ENCODER_REV : INT ;	//SCREW FEEDER ENOCODER REVOLUTION INPUT
   SF1_SPARE_MEMORY_WORD1 : DINT ;
   SF2_PULSE_1 : BOOL ;
   SF2_PULSE_2 : BOOL ;
   SF2_PULSE_3 : BOOL ;
   SF2_PULSE_4 : BOOL ;
   SL_GT_2_OP_CUT : BOOL ;	//SLIDE GATE OPEN OPERATION COMPLETED BIT
   SL_GT_2_CLS_CUT : BOOL ;	//SLIDE GATE CLOSE OPERATION COMPLETED BIT
   SF2_MOTOR_FLT_BIT : BOOL ;	//SCREW FEEDER MOTOR 2 FAULT GENERATED
   SL_GT_2_PULSE3 : BOOL ;	//SLIDE GATE 2 PULSE
   SL_GT_2_OP_TMR : INT ;	//SLIDE GATE OPEN OPERATION COMPLETED TIMER
   SL_GT_2_OP_TIME : INT ;	//SLIDE GATE OPEN OPERATION COMPLETED TIME
   SL_GT_2_CLS_TMR : INT ;	//SLIDE GATE CLOSE OPERATION COMPLETED TIMER
   SL_GT_2_CLS_TIME : INT ;	//SLIDE GATE CLOSE OPERATION COMPLETED TIME
   SF2_FLT_OP_TMR : INT ;	//SCREW FEEDER 2 FAULT OPERATED TIMER
   SF2_FLT_OP_TIME : INT ;	//SCREW FEEDER 2 FAULT OPERATED TIME
   SF2_ENC_PER_REV : DINT ;	//SCREW FEEDER 2 ENCODER PER REVOLUTION
   SF2_HIGH_SPD_COUNT_SET : DINT ;	//SCREW FEEDER 2 HIGH SPEED SET POINT
   SF2_LOW_SPD_COUNT_SET : DINT ;	//SCREW FEEDER 2 LOW SPEED SET POINT
   SF2_HI_SPD_CNT_OVER_BIT : BOOL ;	//SCREW FEEDER 2 HIGH SPEED COUNT OVER
   SF2_LO_SPD_CNT_OVER_BIT : BOOL ;	//SCREW FEEDER 2 LOW SPEED COUNT OVER
   SF2_RST_FOR_LOW_SPD_STA : BOOL ;	//SCREW FEEDER 2 RESET FOR LOW SPEED START
   SL_GT_2_PULSE4 : BOOL ;	//SLIDE GATE 2 PULSE
   SL_GT_2_PULSE1 : BOOL ;	//SLIDE GATE 2 PULSE
   SF2_PULSE : BOOL ;	//SCREW FEEDER 2 PULSE
   SL_GT_2_PULSE2 : BOOL ;	//SLIDE GATE 2 PULSE
   OVEN_CHR_SF2_HI_SPD_STA : BOOL ;	//SCREW FEEDER 2 HIGH SPEED SET IN AUTO
   SF2_PROXI_PULSE : BOOL ;	//SCREW FEEDER 2 PROXIMITY INPUT PULSE
   SF2_HIGH_SPEED_CMD_PF : BOOL ;	//SCREW FEEDER 2 HIGH SPEED COMMAND PROFIBUS
   SF2_LOW_SPEED_CMD_PF : BOOL ;	//SCREW FEEDER 2 LOW SPEED COMMAND PROFIBUS
   SF2_SPARE_MEMORY_BIT8 : BOOL ;	//SCREW FEEDER 2 PULSE USED IN NETWORK 27
   SF2_PULSE_20 : BOOL ;	//SCREW FEEDER 2 PULSE USED IN NETWORK 28
   SF2_PULSE_21 : BOOL ;
   SF2_SPARE_MEMORY_BIT11 : BOOL ;
   SF2_SPARE_MEMORY_BIT12 : BOOL ;
   SF2_SPARE_MEMORY_WORD13 : WORD ;
   SF2_ENCODER_REV : INT ;	//SCREW FEEDER ENOCODER REVOLUTION INPUT
   SF2_SPARE_MEMORY_WORD2 : DINT ;
   SF3_SPARE_MEMORY_BIT : BOOL ;
   SF3_SPARE_MEMORY_BIT1 : BOOL ;
   SF3_SPARE_MEMORY_BIT2 : BOOL ;
   SF3_SPARE_MEMORY_BIT3 : BOOL ;
   SL_GT_3_OP_CUT : BOOL ;	//SLIDE GATE OPEN OPERATION COMPLETED BIT
   SL_GT_3_CLS_CUT : BOOL ;	//SLIDE GATE CLOSE OPERATION COMPLETED BIT
   SF3_MOTOR_FLT_BIT : BOOL ;	//SCREW FEEDER MOTOR 3 FAULT GENERATED
   SL_GT_3_PULSE3 : BOOL ;	//SLIDE GATE 3 PULSE
   SL_GT_3_OP_TMR : INT ;	//SLIDE GATE OPEN OPERATION COMPLETED TIMER
   SL_GT_3_OP_TIME : INT ;	//SLIDE GATE OPEN OPERATION COMPLETED TIME
   SL_GT_3_CLS_TMR : INT ;	//SLIDE GATE CLOSE OPERATION COMPLETED TIMER
   SL_GT_3_CLS_TIME : INT ;	//SLIDE GATE CLOSE OPERATION COMPLETED TIME
   SF3_FLT_OP_TMR : INT ;	//SCREW FEEDER 3 FAULT OPERATED TIMER
   SF3_FLT_OP_TIME : INT ;	//SCREW FEEDER 3 FAULT OPERATED TIME
   SF3_ENC_PER_REV : DINT ;	//SCREW FEEDER 3 ENCODER PER REVOLUTION
   SF3_HIGH_SPD_COUNT_SET : DINT ;	//SCREW FEEDER 3 HIGH SPEED SET POINT
   SF3_LOW_SPD_COUNT_SET : DINT ;	//SCREW FEEDER 3 LOW SPEED SET POINT
   SF3_HI_SPD_CNT_OVER_BIT : BOOL ;	//SCREW FEEDER 3 HIGH SPEED COUNT OVER
   SF3_LO_SPD_CNT_OVER_BIT : BOOL ;	//SCREW FEEDER 3 LOW SPEED COUNT OVER
   SF3_RST_FOR_LOW_SPD_STA : BOOL ;	//SCREW FEEDER 3 RESET FOR LOW SPEED START
   SL_GT_3_PULSE4 : BOOL ;	//SLIDE GATE 3 PULSE
   SL_GT_3_PULSE1 : BOOL ;	//SLIDE GATE 3 PULSE
   SF3_PULSE : BOOL ;	//SCREW FEEDER 3 PULSE
   SL_GT_3_PULSE2 : BOOL ;	//SLIDE GATE 3 PULSE
   OVEN_CHR_SF3_HI_SPD_STA : BOOL ;	//SCREW FEEDER 3 HIGH SPEED SET IN AUTO
   SF3_PROXI_PULSE : BOOL ;	//SCREW FEEDER 3 PROXIMITY INPUT PULSE
   SF3_PULSE_1 : BOOL ;	//SCREW FEEDER 3 PULSE USED IN NETWORK 43
   SF3_PULSE_2 : BOOL ;	//SCREW FEEDER 3 PULSE USED IN NETWORK 44
   SF3_HIGH_SPEED_CMD_PF : BOOL ;	//SCREW FEEDER 3 HIGH SPEED COMMAND PROFIBUS
   SF3_LOW_SPEED_CMD_PF : BOOL ;	//SCREW FEEDER 3 LOW SPEED COMMAND PROFIBUS
   SF3_PULSE_20 : BOOL ;
   SF3_PULSE_21 : BOOL ;
   SF3_SPARE_MEMORY_BIT12 : BOOL ;
   SF3_SPARE_MEMORY_WORD13 : WORD ;
   SF3_ENCODER_REV : INT ;	//SCREW FEEDER ENOCODER REVOLUTION INPUT
   SF3_SPARE_MEMORY_WORD : DINT ;
   SF1_PULSE_30 : BOOL ;
   SF1_PULSE_31 : BOOL ;
   SF1_PULSE_32 : BOOL ;
   SF1_PULSE_33 : BOOL ;
   SF1_PULSE_34 : BOOL ;
   SF1_PULSE_35 : BOOL ;
   SF1_PULSE_36 : BOOL ;
   SF1_PULSE_37 : BOOL ;
   SF1_HI_SPD_CMD_SET : BOOL ;	//SCREW FEEDER 1 HIGH SPEED COMMAND SET
   SF1_LO_SPD_CMD_SET : BOOL ;	//SCREW FEEDER 1 LOW SPEED COMMAND SET
   SF2_HI_SPD_CMD_SET : BOOL ;	//SCREW FEEDER 2 HIGH SPEED COMMAND SET
   SF2_LO_SPD_CMD_SET : BOOL ;	//SCREW FEEDER 2 LOW SPEED COMMAND SET
   SF3_HI_SPD_CMD_SET : BOOL ;	//SCREW FEEDER 3 HIGH SPEED COMMAND SET
   SF3_LO_SPD_CMD_SET : BOOL ;	//SCREW FEEDER 3 LOW SPEED COMMAND SET
   SF1_LO_SPD_CMD_NEG_SET : BOOL ;	//SCREW FEEDER 1 LOW SPEED COMMAND NEGATIVE SET FOR RESISTING ZERO
   SF2_LO_SPD_CMD_NEG_SET : BOOL ;	//SCREW FEEDER 2 LOW SPEED COMMAND NEGATIVE SET FOR RESISTING ZERO
   SF3_LO_SPD_CMD_NEG_SET : BOOL ;	//SCREW FEEDER 3 LOW SPEED COMMAND NEGATIVE SET FOR RESISTING ZERO
  END_STRUCT ;	
BEGIN
   SF_1_RDY_FOR_STA := TRUE;
   SF_2_RDY_FOR_STA := TRUE;
   SF_3_RDY_FOR_STA := TRUE;
   SF_1_STP_PB := TRUE;
   SF_1_HI_SEL := TRUE;
   SF_2_STP_PB := TRUE;
   SF_2_HI_SEL := TRUE;
   SF_3_STP_PB := TRUE;
   SF_3_HI_SEL := TRUE;
   SL_GT_1_OPN_LS := TRUE;
   SF1_FLT_OP_TIME := 5;
   SF1_HIGH_SPD_COUNT_SET := L#56;
   SF1_LOW_SPD_COUNT_SET := L#6;
   SF2_FLT_OP_TIME := 5;
   SF2_HIGH_SPD_COUNT_SET := L#51;
   SF2_LOW_SPD_COUNT_SET := L#6;
   SF3_FLT_OP_TIME := 5;
   SF3_HIGH_SPD_COUNT_SET := L#50;
   SF3_LOW_SPD_COUNT_SET := L#6;
END_DATA_BLOCK

DATA_BLOCK "TATA_COMMUNICATION_DB"	// DB 6
VERSION : 0.1
  STRUCT
   PULSE_1 : BOOL ;	//PULSE 1
   PULSE_2 : BOOL ;	//PULSE 2
   PULSE_3 : BOOL ;	//PULSE 3
   PULSE_4 : BOOL ;	//PULSE 4
   CHAR_COMP_BIT_RESET_TMR : INT ;	//CHARGING COMPLETED BIT TIMER
   CHAR_COMP_BIT_RESET_TM : INT ;	//CHARGING COMPLETED BIT RESET TIME
   TATA_DATA_READ_ERROR : INT ;	//TATA PLC DATA READ ERROR
   TATA_DATA_WRITE_ERROR : INT ;	//TATA PLC DATA WRITE ERROR
  END_STRUCT ;	
BEGIN
   CHAR_COMP_BIT_RESET_TMR := 5;
END_DATA_BLOCK

DATA_BLOCK "INSTANCE DB FOR FM350"	// DB 7
VERSION : 0.1
  STRUCT
   JOB_WR : STRUCT 	// write commands
    NO : BYTE ;	// number
    BUSY : BOOL ;	// job in working
    DONE : BOOL ;	// job is done
    IMPOSS : BOOL ;	// job impossible
    UNKOWN : BOOL ;	// job unkown
   END_STRUCT ;
   JOB_RD : STRUCT 	// read commands
    NO : BYTE ;	// number
    BUSY : BOOL ;	// job in working
    DONE : BOOL ;	// job is done
    IMPOSS : BOOL ;	// job impossible
    UNKOWN : BOOL ;	// job unkown
   END_STRUCT ;
   RESERV_0 : ARRAY  [1 .. 3 ] OF WORD  := 3 (W#16#0) ;	// reserved
   RESERV_1 : WORD ;	// reserved
   MOD_ADR : WORD ;	// module address
   CH_ADR : DWORD ;	// channel address
   DS_OFFS : BYTE ;	// data block offset
   RESERV_2 : BYTE ;	// reserved
   CONTROL_SIGNALS : STRUCT 	// control signals
    BIT0_0 : BOOL ;	// reserved
    BIT0_1 : BOOL ;	// reserved
    BIT0_2 : BOOL ;	// reserved
    BIT0_3 : BOOL ;	// reserved
    BIT0_4 : BOOL ;	// reserved
    BIT0_5 : BOOL ;	// reserved
    BIT0_6 : BOOL ;	// reserved
    BIT0_7 : BOOL ;	// reserved
    CTRL_DQ0 : BOOL ;	// control digital output DQ0
    CTRL_DQ1 : BOOL ;	// control digital output DQ1
    CTRL_DQ2 : BOOL ;	// control digital output DQ2
    CTRL_DQ3 : BOOL ;	// control digital output DQ3
    CTRL_DQ4 : BOOL ;	// control digital output DQ4
    CTRL_DQ5 : BOOL ;	// control digital output DQ5
    CTRL_DQ6 : BOOL ;	// control digital output DQ6
    CTRL_DQ7 : BOOL ;	// control digital output DQ7
    SET_DQ0 : BOOL ;	// set digital output DQ0
    SET_DQ1 : BOOL ;	// set digital output DQ1
    SET_DQ2 : BOOL ;	// set digital output DQ2
    SET_DQ3 : BOOL ;	// set digital output DQ3
    SET_DQ4 : BOOL ;	// set digital output DQ4
    SET_DQ5 : BOOL ;	// set digital output DQ5
    SET_DQ6 : BOOL ;	// set digital output DQ6
    SET_DQ7 : BOOL ;	// set digital output DQ7
    SW_GATE0 : BOOL ;	// software gate 0
    SW_GATE1 : BOOL ;	// software gate 1
    SW_GATE2 : BOOL ;	// software gate 2
    SW_GATE3 : BOOL ;	// software gate 3
    SW_GATE4 : BOOL ;	// software gate 4
    SW_GATE5 : BOOL ;	// software gate 5
    SW_GATE6 : BOOL ;	// software gate 6
    SW_GATE7 : BOOL ;	// software gate 7
    CTRL_DWORD1 : DWORD ;	// reserved
    CTRL_DWORD2 : DWORD ;	// reserved
    CTRL_DWORD3 : DWORD ;	// reserved
   END_STRUCT ;
   CHECKBACK_SIGNALS : STRUCT 	// checkback signals
    BIT0_0 : BOOL ;	// reserved
    STS_TFB : BOOL ;	// status test free bit
    BIT0_2 : BOOL ;	// reserved
    BIT0_3 : BOOL ;	// reserved
    DATA_ERR : BOOL ;	// data error bit
    BIT0_5 : BOOL ;	// reserved
    BIT0_6 : BOOL ;	// reserved
    PARA : BOOL ;	// module parametrized
    STS_CMP0 : BOOL ;	// status compare event 0
    STS_CMP1 : BOOL ;	// status compare event 1
    STS_CMP2 : BOOL ;	// status compare event 2
    STS_CMP3 : BOOL ;	// status compare event 3
    STS_CMP4 : BOOL ;	// status compare event 4
    STS_CMP5 : BOOL ;	// status compare event 5
    STS_CMP6 : BOOL ;	// status compare event 6
    STS_CMP7 : BOOL ;	// status compare event 7
    STS_UFLW0 : BOOL ;	// status counter 0 passed the underflow value
    STS_UFLW1 : BOOL ;	// status counter 1 passed the underflow value
    STS_UFLW2 : BOOL ;	// status counter 2 passed the underflow value
    STS_UFLW3 : BOOL ;	// status counter 3 passed the underflow value
    STS_UFLW4 : BOOL ;	// status counter 4 passed the underflow value
    STS_UFLW5 : BOOL ;	// status counter 5 passed the underflow value
    STS_UFLW6 : BOOL ;	// status counter 6 passed the underflow value
    STS_UFLW7 : BOOL ;	// status counter 7 passed the underflow value
    STS_OFLW0 : BOOL ;	// status counter 0 passed the overflow value
    STS_OFLW1 : BOOL ;	// status counter 1 passed the overflow value
    STS_OFLW2 : BOOL ;	// status counter 2 passed the overflow value
    STS_OFLW3 : BOOL ;	// status counter 3 passed the overflow value
    STS_OFLW4 : BOOL ;	// status counter 4 passed the overflow value
    STS_OFLW5 : BOOL ;	// status counter 5 passed the overflow value
    STS_OFLW6 : BOOL ;	// status counter 6 passed the overflow value
    STS_OFLW7 : BOOL ;	// status counter 7 passed the overflow value
    STS_DIR0 : BOOL ;	// status counter 0 direction
    STS_DIR1 : BOOL ;	// status counter 1 direction
    STS_DIR2 : BOOL ;	// status counter 2 direction
    STS_DIR3 : BOOL ;	// status counter 3 direction
    STS_DIR4 : BOOL ;	// status counter 4 direction
    STS_DIR5 : BOOL ;	// status counter 5 direction
    STS_DIR6 : BOOL ;	// status counter 6 direction
    STS_DIR7 : BOOL ;	// status counter 7 direction
    STS_DI0 : BOOL ;	// status of the digital input 0
    STS_DI1 : BOOL ;	// status of the digital input 1
    STS_DI2 : BOOL ;	// status of the digital input 2
    STS_DI3 : BOOL ;	// status of the digital input 3
    STS_DI4 : BOOL ;	// status of the digital input 4
    STS_DI5 : BOOL ;	// status of the digital input 5
    STS_DI6 : BOOL ;	// status of the digital input 6
    STS_DI7 : BOOL ;	// status of the digital input 7
    STS_DQ0 : BOOL ;	// status of the digital output 0
    STS_DQ1 : BOOL ;	// status of the digital output 1
    STS_DQ2 : BOOL ;	// status of the digital output 2
    STS_DQ3 : BOOL ;	// status of the digital output 3
    STS_DQ4 : BOOL ;	// status of the digital output 4
    STS_DQ5 : BOOL ;	// status of the digital output 5
    STS_DQ6 : BOOL ;	// status of the digital output 6
    STS_DQ7 : BOOL ;	// status of the digital output 7
    STS_GATE0 : BOOL ;	// status of the internal gate 0
    STS_GATE1 : BOOL ;	// status of the internal gate 1
    STS_GATE2 : BOOL ;	// status of the internal gate 2
    STS_GATE3 : BOOL ;	// status of the internal gate 3
    STS_GATE4 : BOOL ;	// status of the internal gate 4
    STS_GATE5 : BOOL ;	// status of the internal gate 5
    STS_GATE6 : BOOL ;	// status of the internal gate 6
    STS_GATE7 : BOOL ;	// status of the internal gate 7
    USER_STAT_WORD0 : WORD ;	// user specific status
    USER_STAT_WORD1 : WORD ;	// user specific status
    USER_STAT_WORD2 : WORD ;	// user specific status
    USER_STAT_WORD3 : WORD ;	// user specific status
   END_STRUCT ;
   LOAD_VAL0 : DINT ;	// load value counter 0
   LOAD_VAL1 : DINT ;	// load value counter 1
   LOAD_VAL2 : DINT ;	// load value counter 2
   LOAD_VAL3 : DINT ;	// load value counter 3
   LOAD_VAL4 : DINT ;	// load value counter 4
   LOAD_VAL5 : DINT ;	// load value counter 5
   LOAD_VAL6 : DINT ;	// load value counter 6
   LOAD_VAL7 : DINT ;	// load value counter 7
   LOAD_PREPARE_VAL0 : DINT ;	// load prepare value counter 0
   LOAD_PREPARE_VAL1 : DINT ;	// load prepare value counter 1
   LOAD_PREPARE_VAL2 : DINT ;	// load prepare value counter 2
   LOAD_PREPARE_VAL3 : DINT ;	// load prepare value counter 3
   LOAD_PREPARE_VAL4 : DINT ;	// load prepare value counter 4
   LOAD_PREPARE_VAL5 : DINT ;	// load prepare value counter 5
   LOAD_PREPARE_VAL6 : DINT ;	// load prepare value counter 6
   LOAD_PREPARE_VAL7 : DINT ;	// load prepare value counter 7
   CMP_VAL0 : DINT ;	// comparator value 0
   CMP_VAL1 : DINT ;	// comparator value 1
   CMP_VAL2 : DINT ;	// comparator value 2
   CMP_VAL3 : DINT ;	// comparator value 3
   CMP_VAL4 : DINT ;	// comparator value 4
   CMP_VAL5 : DINT ;	// comparator value 5
   CMP_VAL6 : DINT ;	// comparator value 6
   CMP_VAL7 : DINT ;	// comparator value 7
   ACT_CNTV0 : DINT ;	// actual counter value 0
   ACT_MSRV0 : DINT ;	// act. measurement value 0
   ACT_CNTV1 : DINT ;	// actual counter value 1
   ACT_MSRV1 : DINT ;	// act. measurement value 1
   ACT_CNTV2 : DINT ;	// actual counter value 2
   ACT_MSRV2 : DINT ;	// act. measurement value 2
   ACT_CNTV3 : DINT ;	// actual counter value 3
   ACT_MSRV3 : DINT ;	// act. measurement value 3
   ACT_CNTV4 : DINT ;	// actual counter value 4
   ACT_MSRV4 : DINT ;	// act. measurement value 4
   ACT_CNTV5 : DINT ;	// actual counter value 5
   ACT_MSRV5 : DINT ;	// act. measurement value 5
   ACT_CNTV6 : DINT ;	// actual counter value 6
   ACT_MSRV6 : DINT ;	// act. measurement value 6
   ACT_CNTV7 : DINT ;	// actual counter value 7
   ACT_MSRV7 : DINT ;	// act. measurement value 7
   DIAGNOSTIC_INT_INFO : STRUCT 	// diagnostic int. information
    BYTE0 : BYTE ;	// byte 0
    BYTE1 : BYTE ;	// byte 1
    BYTE2 : BYTE ;	// byte 2
    BYTE3 : BYTE ;	// byte 3
    BYTE4 : BYTE ;	// channel type info
    BYTE5 : BYTE ;	// channel info length
    BYTE6 : BYTE ;	// number of channels
    BYTE7 : BYTE ;	// channel error vector
    BYTE8 : BYTE ;	// error counter 0
    BYTE9 : BYTE ;	// error counter 1
    BYTE10 : BYTE ;	// error counter 2
    BYTE11 : BYTE ;	// error counter 3
    BYTE12 : BYTE ;	// error counter 4
    BYTE13 : BYTE ;	// error counter 5
    BYTE14 : BYTE ;	// error counter 6
    BYTE15 : BYTE ;	// error counter 7
   END_STRUCT ;
  END_STRUCT ;	
BEGIN
   MOD_ADR := W#16#110;
   CH_ADR := DW#16#880;
END_DATA_BLOCK

DATA_BLOCK "08_LID_MECHANISM_DB"	// DB 8
VERSION : 0.1
  STRUCT
   LID_MECH_REP_MD : BOOL ;	//LID MECHANISM REPAIR MODE
   LID_MECH_OPER_MD : BOOL ;	//LID MECHANISM OPERATING MODE
   LID_MECH_MAN_MD : BOOL ;	//LID MECHANISM MANUAL MODE
   LID_MECH_SA_MD : BOOL ;	//LID MECHANISM SEMI AUTO MODE
   LID_FR_CLN_MTR_1_RDY_STA : BOOL ;	//LID AND FRAME CLEANER 1 READY FOR START
   LID_FR_CLN_MTR_1_RUN_FB : BOOL ;	//LID AND FRAME CLEANER 1 RUN FEEDBACK
   LID_FR_CLN_MTR_1_OLR_TRP : BOOL ;	//LID AND FRAME CLEANER 1 OVERLOAD TRIP
   LID_FR_CLN_MTR_2_RDY_STA : BOOL ;	//LID AND FRAME CLEANER 2 READY FOR START
   LID_FR_CLN_MTR_2_RUN_FB : BOOL ;	//LID AND FRAME CLEANER 2 RUN FEEDBACK
   LID_FR_CLN_MTR_2_OLR_TRP : BOOL ;	//LID AND FRAME CLEANER 2 OVERLOAD TRIP
   LID_FR_CLN_MTR_3_RDY_STA : BOOL ;	//LID AND FRAME CLEANER 3 READY FOR START
   LID_FR_CLN_MTR_3_RUN_FB : BOOL ;	//LID AND FRAME CLEANER 3 RUN FEEDBACK
   LID_FR_CLN_MTR_3_OLR_TRP : BOOL ;	//LID AND FRAME CLEANER 3 OVERLOAD TRIP
   LID_FR_CL_MTR_1_STA_PB : BOOL ;	//LID FRAME CLEANER MOTOR 1 START PUSH BUTTON
   LID_FR_CL_MTR_1_STP_PB : BOOL ;	//LID FRAME CLEANER MOTOR 1 STOP PUSH BUTTON
   LID_FR_CL_MTR_2_STA_PB : BOOL ;	//LID FRAME CLEANER MOTOR 2 START PUSH BUTTON
   LID_FR_CL_MTR_2_STP_PB : BOOL ;	//LID FRAME CLEANER MOTOR 2 STOP PUSH BUTTON
   LID_FR_CL_MTR_3_STA_PB : BOOL ;	//LID FRAME CLEANER MOTOR 3 START PUSH BUTTON
   LID_FR_CL_MTR_3_STP_PB : BOOL ;	//LID FRAME CLEANER MOTOR 3 STOP PUSH BUTTON
   SPARE_5 : BOOL ;
   SPARE_6 : BOOL ;
   LID_LIFT_1_CAR_FWD_STA : BOOL ;	//LID LIFTER 1 CARRIAGE FORWARD START PUSH BUTTON
   LID_LIFT_1_CAR_RET_STA : BOOL ;	//LID LIFTER 1 CARRIAGE RETRACT START PUSH BUTTON
   LID_LIFT_1_VER_DN_STA : BOOL ;	//LID LIFTER 1 VERTICAL DOWN START PUSH BUTTON
   LID_LIFT_1_VER_UP_STA : BOOL ;	//LID LIFTER 1 VERTICAL UP START PUSH BUTTON
   LID_1_FRM_CLNR_DN_STA : BOOL ;	//LID 1 FRAME CLEANER DOWN START
   LID_1_FRM_CLNR_UP_STA : BOOL ;	//LID 1 FRAME CLEANER UP START
   LID_1_TELES_DN_STA_PB : BOOL ;	//LID 1 TELESCOPE DOWN START PUSH BUTTON
   LID_1_TELES_UP_STA_PB : BOOL ;	//LID 1 TELESCOPE UP START PUSH BUTTON
   LID_1_SLI_GT_CLS_STA_PB : BOOL ;	//LID 1 SLIDE GATE CLOSE PUSH BUTTON
   LID_1_SLI_GT_OPN_STA_PB : BOOL ;	//LID 1 SLIDE GATE OPEN PUSH BUTTON
   LID_LIFT_1_CAR_FWD_LS : BOOL ;	//LID LIFTER 1 CARRIAGE FORWARD LIMIT SWITCH
   LID_LIFT_1_CAR_RET_LS : BOOL ;	//LID LIFTER 1 CARRIAGE RETRACT LIMIT SWITCH
   LID_LIFT_1_VER_DN_LS : BOOL ;	//LID LIFTER 1 VERTICAL DOWN LIMIT SWITCH
   LID_LIFT_1_VER_UP_LS : BOOL ;	//LID LIFTER 1 VERTICAL UP LIMIT SWITCH
   TELE_1_DN_LS : BOOL ;	//TELESCOPE 1 DOWN LIMIT SWITCH
   TELE_1_UP_LS : BOOL ;	//TELESCOPE 1 UP LIMIT SWITCH
   SPARE_7 : BOOL ;
   SPARE_8 : BOOL ;
   LID_LIFT_2_CAR_FWD_STA : BOOL ;	//LID LIFTER 2 CARRIAGE FORWARD START PUSH BUTTON
   LID_LIFT_2_CAR_RET_STA : BOOL ;	//LID LIFTER 2 CARRIAGE RETRACT START PUSH BUTTON
   LID_LIFT_2_VER_DN_STA : BOOL ;	//LID LIFTER 2 VERTICAL DOWN START PUSH BUTTON
   LID_LIFT_2_VER_UP_STA : BOOL ;	//LID LIFTER 2 VERTICAL UP START PUSH BUTTON
   LID_2_FRM_CLNR_DN_STA : BOOL ;	//LID 2 FRAME CLEANER DOWN START
   LID_2_FRM_CLNR_UP_STA : BOOL ;	//LID 2 FRAME CLEANER UP START
   LID_2_TELES_DN_STA_PB : BOOL ;	//TELESCOPE 2  DOWN START PUSH BUTTON
   LID_2_TELES_UP_STA_PB : BOOL ;	//TELESCOPE 2 UP START PUSH BUTTON
   LID_2_SLI_GT_CLS_STA_PB : BOOL ;	//LID 2 SLIDE GATE CLOSE PUSH BUTTON
   LID_2_SLI_GT_OPN_STA_PB : BOOL ;	//LID 2 SLIDE GATE OPEN PUSH BUTTON
   LID_LIFT_2_CAR_FWD_LS : BOOL ;	//LID LIFTER 2 CARRIAGE FORWARD LIMIT SWITCH
   LID_LIFT_2_CAR_RET_LS : BOOL ;	//LID LIFTER 2 CARRIAGE RETRACT LIMIT SWITCH
   LID_LIFT_2_VER_DN_LS : BOOL ;	//LID LIFTER 2 VERTICAL DOWN LIMIT SWITCH
   LID_LIFT_2_VER_UP_LS : BOOL ;	//LID LIFTER 2 VERTICAL UP LIMIT SWITCH
   TELE_2_DN_LS : BOOL ;	//TELESCOPE 2 DOWN LIMIT SWITCH
   TELE_2_UP_LS : BOOL ;	//TELESCOPE 2 UP LIMIT SWITCH
   LID_3_CAR_FWD_STA : BOOL ;	//LID 1 CARRIAGE FORWARD START PUSH BUTTON
   LID_3_CAR_RET_STA : BOOL ;	//LID 1 CARRIAGE RETRACT START PUSH BUTTON
   LID_LIFT_3_CAR_FWD_STA : BOOL ;	//LID LIFTER 1 CARRIAGE FORWARD START PUSH BUTTON
   LID_LIFT_3_CAR_RET_STA : BOOL ;	//LID LIFTER 1 CARRIAGE RETRACT START PUSH BUTTON
   LID_LIFT_3_VER_DN_STA : BOOL ;	//LID LIFTER 1 VERTICAL DOWN START PUSH BUTTON
   LID_LIFT_3_VER_UP_STA : BOOL ;	//LID LIFTER 1 VERTICAL UP START PUSH BUTTON
   LID_3_FRM_CLNR_DN_STA : BOOL ;	//LID 1 FRAME CLEANER DOWN START
   LID_3_FRM_CLNR_UP_STA : BOOL ;	//LID 1 FRAME CLEANER UP START
   LID_3_TELES_DN_STA_PB : BOOL ;	//TELESCOPE 3 DOWN START PUSH BUTTON
   LID_3_TELES_UP_STA_PB : BOOL ;	//TELESCOPE 3 UP START PUSH BUTTON
   LID_3_SLI_GT_CLS_STA_PB : BOOL ;	//LID 3 SLIDE GATE CLOSE PUSH BUTTON
   LID_3_SLI_GT_OPN_STA_PB : BOOL ;	//LID 3 SLIDE GATE OPEN PUSH BUTTON
   LID_LIFT_3_CAR_FWD_LS : BOOL ;	//LID LIFTER 3 CARRIAGE FORWARD LIMIT SWITCH
   LID_LIFT_3_CAR_RET_LS : BOOL ;	//LID LIFTER 3 CARRIAGE RETRACT LIMIT SWITCH
   LID_LIFT_3_VER_DN_LS : BOOL ;	//LID LIFTER 3 VERTICAL DOWN LIMIT SWITCH
   LID_LIFT_3_VER_UP_LS : BOOL ;	//LID LIFTER 3 VERTICAL UP LIMIT SWITCH
   TELE_3_DN_LS : BOOL ;	//TELESCOPE 3 DOWN LIMIT SWITCH
   TELE_3_UP_LS : BOOL ;	//TELESCOPE 3 UP LIMIT SWITCH
   LID_OSC_1_ON_CMD : BOOL ;	//LID OSCILLATION 1 ON CMD
   LID_OSC_2_ON_CMD : BOOL ;	//LID OSCILLATION 2 ON CMD
   LID_OSC_3_ON_CMD : BOOL ;	//LID OSCILLATION 3 ON CMD
   LID_OSC_1_ON_IND : BOOL ;	//LID OSCILLATION 1 ON INDICATION
   LID_OSC_2_ON_IND : BOOL ;	//LID OSCILLATION 2 ON INDICATION
   LID_OSC_3_ON_IND : BOOL ;	//LID OSCILLATION 3 ON INDICATION
   LID_FR_CLNR_1_MTR_ON_CMD : BOOL ;	//LID FRAME CLEANER 1 MOTOR ON COMMAND
   LID_FR_CLNR_2_MTR_ON_CMD : BOOL ;	//LID FRAME CLEANER 2 MOTOR ON COMMAND
   LID_FR_CLNR_3_MTR_ON_CMD : BOOL ;	//LID FRAME CLEANER 3 MOTOR ON COMMAND
   LID_FRM_CLNR_1_ON_IND : BOOL ;	//LID FRAME CLEANER 1 ON INDICATION
   LID_FRM_CLNR_2_ON_IND : BOOL ;	//LID FRAME CLEANER 2 ON INDICATION
   LID_FRM_CLNR_3_ON_IND : BOOL ;	//LID FRAME CLEANER 3 ON INDICATION
   LID_LIFT_1_CAR_FWD_CMD : BOOL ;	//LID LIFTER 1 CARRIAGE FORWARD COMMAND
   LID_LIFT_1_CAR_REV_CMD : BOOL ;	//LID LIFTER 1 CARRIAGE REVERSE COMMAND
   LID_LIFT_1_VER_DN_CMD : BOOL ;	//LID LIFTER 1 VERTICAL DOWN COMMAND
   LID_LIFT_1_VER_UP_CMD : BOOL ;	//LID LIFTER 1 VERTICAL UP COMMAND
   LID_FRM_CLNR_1_DN_CMD : BOOL ;	//LID FRAME CLEANER 1 DOWN COMMAND
   LID_FRM_CLNR_1_UP_CMD : BOOL ;	//LID FRAME CLEANER 1 UP COMMAND
   TELE_1_DN_CMD : BOOL ;	//TELESCOPE 1 DOWN COMMAND
   TELE_1_UP_CMD : BOOL ;	//TELESCOPE 1 UP COMMAND
   LID_LIFT_1_CAR_FWD_IND : BOOL ;	//LID LIFTER 1 CARRIAGE FORWARD ON INDICATION
   LID_LIFT_1_CAR_RET_IND : BOOL ;	//LID LIFTER 1 CARRIAGE RETRACT ON INDICATION
   LID_LIFT_1_VER_DN_IND : BOOL ;	//LID LIFTER 1 VERTICAL DOWN ON INDICATION
   LID_LIFT_1_VER_UP_IND : BOOL ;	//LID LIFTER 1 VERTICAL UP ON INDICATION
   LID_LIFT_1_CLNR_POS_IND : BOOL ;	//LID LIFTER 1 CLEANING POSITION ON INDICATION
   LID_FRM_CLNR_1_DN_IND : BOOL ;	//LID FRAME CLEANER 1 DOWN INDICATION
   LID_FRM_CLNR_1_UP_IND : BOOL ;	//LID FRAME CLEANER 1 UP INDICATION
   TELE_1_DN_IND : BOOL ;	//TELESCOPE 1 DOWN INDICATION
   TELE_1_UP_IND : BOOL ;	//TELESCOPE 1 UP INDICATION
   LID_LIFT_2_CAR_FWD_CMD : BOOL ;	//LID LIFTER 2 CARRIAGE FORWARD COMMAND
   LID_LIFT_2_CAR_REV_CMD : BOOL ;	//LID LIFTER 2 CARRIAGE REVERSE COMMAND
   LID_LIFT_2_VER_DN_CMD : BOOL ;	//LID LIFTER 2 VERTICAL DOWN COMMAND
   LID_LIFT_2_VER_UP_CMD : BOOL ;	//LID LIFTER 2 VERTICAL UP COMMAND
   LID_FRM_CLNR_2_DN_CMD : BOOL ;	//LID FRAME CLEANER 2 DOWN COMMAND
   LID_FRM_CLNR_2_UP_CMD : BOOL ;	//LID FRAME CLEANER 2 UP COMMAND
   TELE_2_DN_CMD : BOOL ;	//TELESCOPE 2 DOWN COMMAND
   TELE_2_UP_CMD : BOOL ;	//TELESCOPE 2 UP COMMAND
   LID_LIFT_2_CAR_FWD_IND : BOOL ;	//LID LIFTER 2 CARRIAGE FORWARD ON INDICATION
   LID_LIFT_2_CAR_RET_IND : BOOL ;	//LID LIFTER 2 CARRIAGE RETRACT ON INDICATION
   LID_LIFT_2_VER_DN_IND : BOOL ;	//LID LIFTER 2 VERTICAL DOWN ON INDICATION
   LID_LIFT_2_VER_UP_IND : BOOL ;	//LID LIFTER 2 VERTICAL UP ON INDICATION
   LID_LIFT_2_CLNR_POS_IND : BOOL ;	//LID LIFTER 2 CLEANING POSITION ON INDICATION
   LID_FRM_CLNR_2_DN_IND : BOOL ;	//LID FRAME CLEANER 2 DOWN INDICATION
   LID_FRM_CLNR_2_UP_IND : BOOL ;	//LID FRAME CLEANER 2 UP INDICATION
   TELE_2_DN_IND : BOOL ;	//TELESCOPE 2 DOWN INDICATION
   TELE_2_UP_IND : BOOL ;	//TELESCOPE 2 UP INDICATION
   LID_LIFT_3_CAR_FWD_CMD : BOOL ;	//LID LIFTER 3 CARRIAGE FORWARD COMMAND
   LID_LIFT_3_CAR_REV_CMD : BOOL ;	//LID LIFTER 3 CARRIAGE REVERSE COMMAND
   LID_LIFT_3_VER_DN_CMD : BOOL ;	//LID LIFTER 3 VERTICAL DOWN COMMAND
   LID_LIFT_3_VER_UP_CMD : BOOL ;	//LID LIFTER 3 VERTICAL UP COMMAND
   LID_FRM_CLNR_3_DN_CMD : BOOL ;	//LID FRAME CLEANER 2 DOWN COMMAND
   LID_FRM_CLNR_3_UP_CMD : BOOL ;	//LID FRAME CLEANER 3 UP COMMAND
   TELE_3_DN_CMD : BOOL ;	//TELESCOPE 3 DOWN COMMAND
   TELE_3_UP_CMD : BOOL ;	//TELESCOPE 3 UP COMMAND
   LID_LIFT_3_CAR_FWD_IND : BOOL ;	//LID LIFTER 3 CARRIAGE FORWARD ON INDICATION
   LID_LIFT_3_CAR_RET_IND : BOOL ;	//LID LIFTER 3 CARRIAGE RETRACT ON INDICATION
   LID_LIFT_3_VER_DN_IND : BOOL ;	//LID LIFTER 3 VERTICAL DOWN ON INDICATION
   LID_LIFT_3_VER_UP_IND : BOOL ;	//LID LIFTER 3 VERTICAL UP ON INDICATION
   LID_LIFT_3_CLNR_POS_IND : BOOL ;	//LID LIFTER 3 CLEANING POSITION ON INDICATION
   LID_FRM_CLNR_3_DN_IND : BOOL ;	//LID FRAME CLEANER 3 DOWN INDICATION
   LID_FRM_CLNR_3_UP_IND : BOOL ;	//LID FRAME CLEANER 3 UP INDICATION
   TELE_3_DN_IND : BOOL ;	//TELESCOPE 3 DOWN INDICATION
   TELE_3_UP_IND : BOOL ;	//TELESCOPE 3 UP INDICATION
   LID_INTERLOCK : BOOL ;	//LID MECHANISM MAIN INTERLOCK
   PULSE_1 : BOOL ;
   PULSE_2 : BOOL ;
   PULSE_3 : BOOL ;
   PULSE_4 : BOOL ;
   PULSE_5 : BOOL ;
   PULSE_6 : BOOL ;
   PULSE_7 : BOOL ;
   LID_FR_CLN_1_MTR_FLT_TIM : INT ;
   LID_FR_CLN_1_MTR_FLT_SET : INT ;
   LID_FR_CLN_1_MTR_FB_FLT : BOOL ;
   LID_LIFT_1_CLN_LS : BOOL ;	//LID LIFTER 1 CLEANING LIMIT SWITCH
   LID_FRM_CLNR_1_DN_LS : BOOL ;	//LID FRAME CLEANER 1 DOWN LIMIT SWITCH
   LID_FRM_CLNR_1_UP_LS : BOOL ;	//LID FRAME CLEANER 1 UP LIMIT SWITCH
   LID_LIFT_2_CLN_LS : BOOL ;	//LID LIFTER 2 CLEANING LIMIT SWITCH
   LID_FRM_CLNR_2_DN_LS : BOOL ;	//LID FRAME 2 CLEANING DOWN LIMIT SWITCH
   LID_FRM_CLNR_2_UP_LS : BOOL ;	//LID FRAME 2 CLEANING UP LIMIT SWITCH
   LID_LIFT_3_CLN_LS : BOOL ;	//LID LIFTER 3 CLEANING LIMIT SWITCH
   LID_FRM_CLNR_3_DN_LS : BOOL ;	//LID FRAME CLEANER 3 DOWN LIMIT SWITCH
   LID_FRM_CLNR_3_UP_LS : BOOL ;	//LID FRAME CLEANER 3 UP LIMIT SWITCH
   PREP_TO_CHARGE_PB : BOOL ;	//PREPARE TO CHARGE PUSH BUTTON CD
   FIN_CHARGE_PB : BOOL ;	//FINISH CHARGING PUSH BUTTON CD
   MAG_1_ENER_FB : BOOL ;	//MAGNET 1 ENERGISED FEEDBACK
   MAG_2_ENER_FB : BOOL ;	//MAGNET 2 ENERGISED FEEDBACK
   MAG_3_ENER_FB : BOOL ;	//MAGNET 3 ENERGISED FEEDBACK
   MAG_1_STA_PB : BOOL ;	//MAGNET 1 START PUSH BUTTON
   MAG_2_STA_PB : BOOL ;	//MAGNET 2 START PUSH BUTTON
   MAG_3_STA_PB : BOOL ;	//MAGNET 3 START PUSH BUTTON
   MAG_1_STP_PB : BOOL ;	//MAGNET 1 STOP PUSH BUTTON
   MAG_2_STP_PB : BOOL ;	//MAGNET 2 STOP PUSH BUTTON
   MAG_3_STP_PB : BOOL ;	//MAGNET 3 STOP PUSH BUTTON
   LID_1_MAG_LS : BOOL ;	//LID 1 AT MAGNETIC LIMIT SWITCH
   LID_2_MAG_LS : BOOL ;	//LID 2 AT MAGNETIC LIMIT SWITCH
   LID_3_MAG_LS : BOOL ;	//LID 3 AT MAGNETIC LIMIT SWITCH
   LID_1_OSC_MTR_RDY_STA : BOOL ;	//LID 1 OSCILLATION MOTOR READY FOR START
   LID_1_OSC_MTR_RUN_FB : BOOL ;	//LID 1 OSCILLATION MOTOR RUN FEEDBACK
   LID_1_OSC_OLR_TRIP : BOOL ;	//LID 1 OSCILLATION MOTOR OVERLOAD TRIP
   LID_2_OSC_MTR_RDY_STA : BOOL ;	//LID 2 OSCILLATION MOTOR READY FOR START
   LID_2_OSC_MTR_RUN_FB : BOOL ;	//LID 2 OSCILLATION MOTOR RUN FEEDBACK
   LID_2_OSC_OLR_TRIP : BOOL ;	//LID 2 OSCILLATION MOTOR OVERLOAD TRIP
   LID_3_OSC_MTR_RDY_STA : BOOL ;	//LID 3 OSCILLATION MOTOR READY FOR START
   LID_3_OSC_MTR_RUN_FB : BOOL ;	//LID 3 OSCILLATION MOTOR RUN FEEDBACK
   LID_3_OSC_OLR_TRIP : BOOL ;	//LID 3 OSCILLATION MOTOR OVERLOAD TRIP
   LID_1_OSC_MTR_STA_PB : BOOL ;	//LID 1 OSCILLATION MOTOR START PUSH BUTTON
   LID_1_OSC_MTR_STP_PB : BOOL ;	//LID 1 OSCILLATION MOTOR STOP PUSH BUTTON
   LID_2_OSC_MTR_STA_PB : BOOL ;	//LID 2 OSCILLATION MOTOR START PUSH BUTTON
   LID_2_OSC_MTR_STP_PB : BOOL ;	//LID 2 OSCILLATION MOTOR STOP PUSH BUTTON
   LID_3_OSC_MTR_STA_PB : BOOL ;	//LID 3 OSCILLATION MOTOR START PUSH BUTTON
   LID_3_OSC_MTR_STP_PB : BOOL ;	//LID 3 OSCILLATION MOTOR STOP PUSH BUTTON
   MAG_1_ON_CMD : BOOL ;	//LID 1 MAGNET ON COMMAND
   MAG_2_ON_CMD : BOOL ;	//LID 2 MAGNET ON COMMAND
   MAG_3_ON_CMD : BOOL ;	//LID 3 MAGNET ON COMMAND
   MAGNET_ON_CMD : BOOL ;	//MAGNET ON COMMAND
   MAG_1_ON_IND : BOOL ;	//LID 1 MAGNET ON INDICATION
   MAG_2_ON_IND : BOOL ;	//LID 2 MAGNET ON INDICATION
   MAG_3_ON_IND : BOOL ;	//LID 3 MAGNET ON INDICATION
   LID_AT_MAG_1_ON_IND : BOOL ;	//LID 1 AT MAGNET ON INDICATION
   LID_AT_MAG_2_ON_IND : BOOL ;	//LID 2 AT MAGNET ON INDICATION
   LID_AT_MAG_3_ON_IND : BOOL ;	//LID 3 AT MAGNET ON INDICATION
   DC_PWR_PCK_RDY_FOR_STA : BOOL ;	//DC POWER READY FOR START
   DC_PWR_PCK_RUN_FB : BOOL ;	//DC POWER PACK RUN FEEDBACK
   LID_OSC_1_LS : BOOL ;	//LID OSCILLATION 1 LIMIT SWITCH
   LID_OSC_2_LS : BOOL ;	//LID OSCILLATION 2 LIMIT SWITCH
   LID_OSC_3_LS : BOOL ;	//LID OSCILLATION 3 LIMIT SWITCH
   MAGNET_FB_FLT : BOOL ;	//MAGNET FEEDBACK FAULT
   MAGNET_FB_FLT_TIME : INT ;	//MAGNET FEEDBACK FAULT TIME
   PREP_TO_CHRG_SET_BIT : BOOL ;	//PREPARE TO CHARGE AUTO SET BIT
   AUTO_STP_SET_BIT : BOOL ;	//AUTO STOP SET BIT
   PREP_TO_CHAR_PB : BOOL ;	//PREPARE TO CHARGE PB FOR AUTO SEQ
   LID_1_CAR_FWD_OP_CUT : BOOL ;	//AUTO CARRIAGE 1 FORWARD COMMAND OPERATION COMPLETE
   LID_1_VER_DN_OP_CUT : BOOL ;	//AUTO VERTICAL 1 DOWN COMMAND OPERATION COMPLETE
   LID_1_MAG_ENER_OP_CUT : BOOL ;	//AUTO MAGNET 1 ENERGISED COMMAND OPERATION COMPLETE
   LID_1_VER_UP_OP_CUT : BOOL ;	//AUTO VERTICAL UP COMMAND OPERATION COMPLETE
   LID_1_CAR_RET_OP_CUT : BOOL ;	//AUTO CARRIAGE 1 RETRACT OPERATION COMPLETE
   LID_1_TEL_DN_OP_CUT : BOOL ;	//AUTO TELESCOPE 1 DOWN OPERATION COMPLETE
   LID_FRM_CLNR_BYPASS : BOOL ;	//LID FRAME CLEANER BYPASS
   LID_1_OSC_CMD_OP_CUT : BOOL ;	//LID OSCILLATION ON COMMAND
   LID_FR_CLN_2_MTR_FB_FLT : BOOL ;
   LID_1_CAR_FWD_OP_CUT_TIM : INT ;	//LID 1 CARRIAGE FORWARD OPERATION COMPLETE TIME
   LID_1_VER_DN_OP_CUT_TIME : INT ;	//LID 1 VERTICAL DOWN OPERATION COMPLETE TIME
   LID_1_MAG_ENER_OVER_TIME : INT ;	//LID 1 MAGNET ENERGIZED OPERATION COMPLETE TIME
   LID_1_VER_UP_OP_CUT_TIM : INT ;	//AUTO VERTICAL UP 1 COMMAND OPERATION COMPLETE TIME
   LID_1_CAR_RET_OP_CUT_TIM : INT ;	//AUTO CARRIAGE 1 RETRACT OPERATION COMPLETE TIME
   LID_1_OSC_CMD_OP_CUT_TIM : INT ;	//LID 1 OSCILLATION COMMAND OPERATION COMPLETE TIME
   LID_FR_CLN_2_MTR_FLT_TIM : INT ;	//LID FRAME CLEANER 2 MOTOR FAULT TIME
   LID_FR_CLN_2_MTR_FLT_SET : INT ;	//LID FRAME CLEANER 2 MOTOR FAULT TIME SET
   LID_2_CAR_FWD_OP_CUT_TIM : INT ;
   LID_2_VER_DN_OP_CUT_TIME : INT ;
   LID_2_MAG_ENER_OP_CUT_TI : INT ;
   LID_2_VER_UP_OP_CUT_TIM : INT ;	//AUTO VERTICAL UP 2 COMMAND OPERATION COMPLETE TIME
   LID_2_CAR_RET_OP_CUT_TIM : INT ;	//AUTO CARRIAGE 2 RETRACT OPERATION COMPLETE TIME
   LID_2_OSC_CMD_OP_CUT_TIM : INT ;	//AUTO OSCIALLATION 2 COMMAND OPERATION COMPLETE TIME
   LID_2_CAR_FWD_OP_CUT : BOOL ;	//AUTO CARRIAGE 2 FORWARD COMMAND OPERATION COMPLETE
   LID_2_VER_DN_OP_CUT : BOOL ;	//AUTO VERTICAL 2 DOWN COMMAND OPERATION COMPLETE
   LID_2_MAG_ENER_OP_CUT : BOOL ;	//AUTO MAGNET 2 ENERGISED COMMAND OPERATION COMPLETE
   LID_2_VER_UP_OP_CUT : BOOL ;	//AUTO VERTICAL UP COMMAND OPERATION COMPLETE
   LID_2_CAR_RET_OP_CUT : BOOL ;	//AUTO CARRIAGE 2 RETRACT OPERATION COMPLETE
   LID_2_TEL_DN_OP_CUT : BOOL ;	//AUTO TELESCOPE 2 DOWN OPERATION COMPLETE
   LID_2_OSC_CMD_OP_CUT : BOOL ;	//LID OSCILLATION ON COMMAND
   PULSE_8 : BOOL ;
   PULSE_9 : BOOL ;
   PULSE_10 : BOOL ;
   PULSE_11 : BOOL ;
   PULSE_12 : BOOL ;
   PULSE_13 : BOOL ;
   PULSE_14 : BOOL ;
   PULSE_15 : BOOL ;
   PULSE_16 : BOOL ;
   LID_FR_CLN_3_MTR_FLT_TIM : INT ;
   LID_FR_CLN_3_MTR_FLT_SET : INT ;
   LID_3_CAR_FWD_OP_CUT_TIM : INT ;
   LID_3_VER_DN_OP_CUT_TIME : INT ;
   LID_3_MAG_ENER_OP_CUT_TI : INT ;
   LID_3_VER_UP_OP_CUT_TIM : INT ;	//AUTO VERTICAL UP 3 COMMAND OPERATION COMPLETE TIME
   LID_3_CAR_RET_OP_CUT_TIM : INT ;	//AUTO CARRIAGE 3 RETRACT OPERATION COMPLETE TIME
   LID_3_OSC_CMD_OP_CUT_TIM : INT ;	//LD 3 OSCILLATION COMMAND OPERATION COMPLETE TIME
   LID_3_CAR_FWD_OP_CUT : BOOL ;	//AUTO CARRIAGE 3 FORWARD COMMAND OPERATION COMPLETE
   LID_3_VER_DN_OP_CUT : BOOL ;	//AUTO VERTICAL 3 DOWN COMMAND OPERATION COMPLETE
   LID_3_MAG_ENER_OP_CUT : BOOL ;	//AUTO MAGNET 3 ENERGISED COMMAND OPERATION COMPLETE
   LID_3_VER_UP_OP_CUT : BOOL ;	//AUTO VERTICAL UP COMMAND OPERATION COMPLETE
   LID_3_CAR_RET_OP_CUT : BOOL ;	//AUTO CARRIAGE 3 RETRACT OPERATION COMPLETE
   LID_3_TEL_DN_OP_CUT : BOOL ;	//AUTO TELESCOPE 3 DOWN OPERATION COMPLETE
   LID_3_OSC_CMD_OP_CUT : BOOL ;	//LID OSCILLATION ON COMMAND
   LID_FR_CLN_3_MTR_FB_FLT : BOOL ;
   PULSE_17 : BOOL ;
   PULSE_18 : BOOL ;
   PULSE_19 : BOOL ;
   PULSE_20 : BOOL ;
   PULSE_21 : BOOL ;
   PULSE_22 : BOOL ;
   PULSE_23 : BOOL ;
   PULSE_24 : BOOL ;
   LID_1_FRM_CLN_DOWN_OP_CU : BOOL ;
   LID_1_FRM_CLN_MTR_ON_OVR : BOOL ;
   LID_LIFT_1_CAR_REV_OP_CU : BOOL ;
   LID_LIFT_1_VER_UP_OP_CUT : BOOL ;
   LID_CAR_2_RET_CMD_OP_CUT : BOOL ;
   LID_FRM_CLNR_2_OP_CUT : BOOL ;
   LID_LIFT_2_CAR_FWD_OP_CU : BOOL ;
   LID_FR_CLNR_2_MTR_ON_OVR : BOOL ;
   LID_OSC_1_ON_FB_FLT_RSET : BOOL ;
   LID_OSC_2_ON_FB_FLT_RSET : BOOL ;
   LID_OSC_3_ON_FB_FLT_RSET : BOOL ;
   FIN_CHARGE_PB_AUTO_SET : BOOL ;	//FINISH CHARGING PUSH BUTTON AUTO SET BIT
   SL_GT_1_CLS_CMD_OP_CUT : BOOL ;	//SLIDE GATE 1 CLOSE COMMAND OPERATION COMPLETE
   TELE_1_UP_CMD_OP_CUT : BOOL ;	//TELESCOPE 1 UP COMMAND OPERATION COMPLETE
   LID_CAR_1_FWD_CMD_OP_CUT : BOOL ;	//LID CARRIAGE 1 FORWARD COMMAND OPERATION COMPLETE
   LID_1_VER_DN_CMD_OP_CUT : BOOL ;	//FINISH CHARING LID VERTICAL 1 DOWN COMMAND OPERATION COMPLETE
   LID_1_VER_UP_CMD_OP_CUT : BOOL ;	//LID VERTICAL 1 UP COMMAND OPERATION COMPLETE
   FIN_CHRG_1_SEQ_OP_CUT : BOOL ;	//LID 1 FINISH CHARGING SEQUENCE OPERATION COMPLETE
   LID_2_VER_DN_CMD_OP_CUT : BOOL ;
   LID_LIFT_3_CAR_FWD_OP_CU : BOOL ;
   LID_1_PROG_IND : BOOL ;	//LID 1 MECHANISM IN PROGRESS
   LID_2_PROG_IND : BOOL ;	//LID 2 MECHANISM IN PROGRESS
   LID_3_PROG_IND : BOOL ;	//LID 3 MECHANISM IN PROGRESS
   SL_GT_2_CLS_CMD_OP_CUT : BOOL ;
   SL_GT_3_CLS_CMD_OP_CUT : BOOL ;
   TELE_2_UP_CMD_OP_CUT : BOOL ;	//TELESCOPE 2 UP COMMAND OPERATION COMPLETE
   LID_2_CAR_FWD_CMD_OP_CUT : BOOL ;
   FC_LID_2_VER_DN_CMD_OP_C : BOOL ;
   FC_LID_2_VER_UP_CMD_OP_C : BOOL ;
   FIN_CHRG_2_SEQ_OP_CUT : BOOL ;	//LID 2 FINISH CHARGING SEQUENCE OPERATION COMPLETE
   TELE_3_UP_CMD_OP_CUT : BOOL ;	//TELESCOPE 3 UP COMMAND OPERATION COMPLETE
   LID_3_CAR_FWD_CMD_OP_CUT : BOOL ;	//FINISH CHARGING LID 3 CARRIAGE FORWARD COMMAND OPERATION COMPLETE
   FC_LID_3_VER_DN_CMD_OP_C : BOOL ;	//FINISH CHARGING LID 3 VERTICAL DOWN COMMAND OPERATION COMPLETE
   FC_LID_3_VER_UP_CMD_OP_C : BOOL ;	//FINISH CHARGING LID 3 VERTICAL UP COMMAND OPERATION COMPLETE
   FIN_CHRG_3_SEQ_OP_CUT : BOOL ;	//LID 3 FINISH CHARGING SEQUENCE OPERATION COMPLETE
   LFC_CAR_1_RET_OP_CUT : BOOL ;	//LID FRAME CLEANER BYPASS SEQUENCE CARRIAGE 1 RETRACT OPERATION COMPLETE
   LFC_FRM_CLN_1_DN_OP_CUT : BOOL ;	//LID FRAME CLEANER BYPASS SEQUENCE FRAME CLEANER 1 DOWN OPERATION COMPLETE
   LFC_CAR_1_FWD_OP_CUT : BOOL ;	//LID FRAME CLEANER BYPASS SEQUENCE CARRIAGE 1 FORWARD OPERATION COMPLETE
   LFC_VER_DN_1_OP_CUT : BOOL ;	//LID FRAME CLEANER BYPASS SEQUENCE VERTICAL DOWN 1 OPERATION COMPLETE
   LFC_MTR_1_ON_OP_CUT : BOOL ;	//LID FRAME CLEANER BYPASS SEQUENCE MOTOR 1 COMMAND OPERATION COMPLETE
   LFC_VER_UP_1_OP_CUT : BOOL ;	//LID FRAME CLEANER BYPASS SEQUENCE VERTICAL UP 1 OPERATION COMPLETE
   LID_FRM_CLNR_1_UP_OP_CUT : BOOL ;	//LID FRAME CLEANER BYPASS SEQUENCE FRAME CLEANER UP 1 OPERATION COMPLETE
   LFC_CAR_2_RET_OP_CUT : BOOL ;	//LID FRAME CLEANER BYPASS SEQUENCE CARRIAGE 2 RETRACT OPERATION COMPLETE
   LFC_FRM_CLN_2_DN_OP_CUT : BOOL ;	//LID FRAME CLEANER BYPASS SEQUENCE FRAME CLEANER 2 DOWN OPERATION COMPLETE
   LFC_CAR_2_FWD_OP_CUT : BOOL ;	//LID FRAME CLEANER BYPASS SEQUENCE CARRIAGE 2 FORWARD OPERATION COMPLETE
   LFC_VER_DN_2_OP_CUT : BOOL ;	//LID FRAME CLEANER BYPASS SEQUENCE VERTICAL DOWN 2 OPERATION COMPLETE
   LFC_MTR_2_ON_OP_CUT : BOOL ;	//LID FRAME CLEANER BYPASS SEQUENCE MOTOR 2 COMMAND OPERATION COMPLETE
   LFC_VER_UP_2_OP_CUT : BOOL ;	//LID FRAME CLEANER BYPASS SEQUENCE VERTICAL UP 2 OPERATION COMPLETE
   LID_FRM_CLNR_2_UP_OP_CUT : BOOL ;	//LID FRAME CLEANER BYPASS SEQUENCE FRAME CLEANER UP 2 OPERATION COMPLETE
   LFC_CAR_3_RET_OP_CUT : BOOL ;	//LID FRAME CLEANER BYPASS SEQUENCE CARRIAGE 3 RETRACT OPERATION COMPLETE
   LFC_FRM_CLN_3_DN_OP_CUT : BOOL ;	//LID FRAME CLEANER BYPASS SEQUENCE FRAME CLEANER 3 DOWN OPERATION COMPLETE
   LFC_CAR_3_FWD_OP_CUT : BOOL ;	//LID FRAME CLEANER BYPASS SEQUENCE CARRIAGE 3 FORWARD OPERATION COMPLETE
   LFC_VER_DN_3_OP_CUT : BOOL ;	//LID FRAME CLEANER BYPASS SEQUENCE VERTICAL DOWN 3 OPERATION COMPLETE
   LFC_MTR_3_ON_OP_CUT : BOOL ;	//LID FRAME CLEANER BYPASS SEQUENCE MOTOR 3 COMMAND OPERATION COMPLETE
   LFC_VER_UP_3_OP_CUT : BOOL ;	//LID FRAME CLEANER BYPASS SEQUENCE VERTICAL UP 3 OPERATION COMPLETE
   LID_FRM_CLNR_3_UP_OP_CUT : BOOL ;	//LID FRAME CLEANER BYPASS SEQUENCE FRAME CLEANER UP 3 OPERATION COMPLETE
   BOOST_1_ON_CMD : BOOL ;	//BOOSTER 1 ON COMMAND
   BOOST_2_ON_CMD : BOOL ;	//BOOSTER 2 ON COMMAND
   BOOST_3_ON_CMD : BOOL ;	//BOOSTER 3 ON COMMAND
   LID_1_STP_PB : BOOL ;	//LID 1 STOP PUSH BUTTON
   LID_2_STP_PB : BOOL ;	//LID 2 STOP PUSH BUTTON
   LID_3_STP_PB : BOOL ;	//LID 3 STOP PUSH BUTTON
  END_STRUCT ;	
BEGIN
   LID_FR_CLN_1_MTR_FLT_SET := 5;
   LID_FR_CLN_2_MTR_FLT_SET := 5;
   LID_FR_CLN_3_MTR_FLT_SET := 5;
END_DATA_BLOCK

DATA_BLOCK "CMD_FROM_TATA"	// DB 10
VERSION : 0.1
  STRUCT
   CC_OnBord_STATUS_BIT : STRUCT
    CC_CHARG_PERM : BOOL ;	//charging interlock OK
    CC_CHARG_LT_MODE : BOOL ;	//Long travel in auto or in man
    CC_TRAVEL_FWD : BOOL ;	//FWD over profibus
    CC_TRAVEL_REV : BOOL ;	//REV over profibus
    CC_TRAVEL_START : BOOL ;	//START over profibus
    CC_TRAVEL_STOP : BOOL ;	//STOP  over profibus
    SpareBit_1 : BOOL ;
    SpareBit_2 : BOOL ;
    SpareBit_3 : BOOL ;
    SpareBit_4 : BOOL ;
    SpareBit_5 : BOOL ;
    SpareBit_6 : BOOL ;
    SpareBit_7 : BOOL ;
    SpareBit_8 : BOOL ;
    SpareBit_9 : BOOL ;
    SpareBit_10 : BOOL ;
    CC_SPEED_REF : INT ;	//Reserve for LT motion (spd_ref) over profibus
    SATA : ARRAY  [1 .. 7 ] OF INT ;
   END_STRUCT ;
  END_STRUCT ;	
BEGIN
END_DATA_BLOCK

DATA_BLOCK "FB_TO_TATA"	// DB 11
VERSION : 0.1
  STRUCT
   CC_MACHINE_STATUS_BIT : STRUCT
    CC_CHARGING_START : BOOL ;
    CC_CHARGING_COMPLET : BOOL ;
    CC_STATU : BOOL ;
    CC_STRT_LEVLING : BOOL ;
    CC_STOP_LEVLING : BOOL ;
    CC_DRV_REV : BOOL ;
    CC_DRV_FWD : BOOL ;
    CC_DRV_STATUS : BOOL ;	//Drive healthy/unhealthy
    CC_PERM : BOOL ;
    SpareBit_2 : BOOL ;
    SpareBit_3 : BOOL ;
    SpareBit_4 : BOOL ;
    SpareBit_5 : BOOL ;
    SpareBit_6 : BOOL ;
    SpareBit_7 : BOOL ;
    CC_SPEED : REAL ;	//CC speed
    Spare_Int0 : INT ;
    Spare_Int1 : INT ;
    SATA : ARRAY  [1 .. 4 ] OF INT ;
   END_STRUCT ;
  END_STRUCT ;	
BEGIN
END_DATA_BLOCK

DATA_BLOCK "WINCC_DB"	// DB 15
VERSION : 0.1
  STRUCT
   MAIN_POWER_ON_PB : BOOL ;	//MAIN_POWER_ON_PB
   MAIN_POWER_OFF_PB : BOOL ;	//MAIN_POWER_OFF_PB
   LAMP_TEST_PB : BOOL ;	//LAMP_TEST_PB
   CONTROL_SELECTION_SS : BOOL ;	//CONTROL_SELECTION_SS
   ALARM_ACK : BOOL ;	//ALARM_ACK
   HYD_LAMP_TEST : BOOL ;
   HYD_ALARM_ACK : BOOL ;
   HYD_CD_LCS_SS_1_2 : BOOL ;
   HYD_PUMP_1_STA_PB : BOOL ;
   HYD_PUMP_1_STOP_PB : BOOL ;
   HYD_PUMP_2_STA_PB : BOOL ;
   HYD_PUMP_2_STOP_PB : BOOL ;
   HYD_HEATER_STA_PB : BOOL ;
   HYD_HEATER_STOP_PB : BOOL ;
   HYD_REPAIR_MODE : BOOL ;
   HYD_MANUAL_MODE : BOOL ;
   HYD_SEMI_AUTO_MODE : BOOL ;
   CONTROL_SELECTION : BOOL ;
   HYD_PUMP_SS : BOOL ;
   HYD_ACCU_STA_PB : BOOL ;
   HYD_ACCU_STOP_PB : BOOL ;
   SIREN_ON_PB : BOOL ;
   SF_1_LAMP_TEST : BOOL ;
   SF_1_ALARM_ACK : BOOL ;
   SF_1_EMERGENCY_STOP : BOOL ;
   SF_1_STA_PB : BOOL ;
   SF_1_STOP_PB : BOOL ;
   SF_1_HIGH_SPEED_SEL : BOOL ;
   SF_1_LOW_SPEED_SEL : BOOL ;
   SF_1_REPAIR_MODE : BOOL ;
   SF_1_MANUAL_MODE : BOOL ;
   SF_1_SEMI_AUTO_MODE : BOOL ;
   SF_1_MACRO_SELECTION : BOOL ;
   SF_2_STOP_PB : BOOL ;
   SF_2_HIGH_SPEED_SEL : BOOL ;
   SF_2_LOW_SPEED_SEL : BOOL ;
   SF_2_LT_OVEN_CHARGE_STA : BOOL ;
   SF_2_LT_SF_SELECTION : BOOL ;
   SF_2_REPAIR_MODE : BOOL ;
   SF_2_MANUAL_MODE : BOOL ;
   SF_2_SEMI_AUTO_MODE : BOOL ;
   SF_2_MACRO_SELECTION : BOOL ;
   SF_2_LAMP_TEST : BOOL ;
   SF_2_ALARM_ACK : BOOL ;
   SF_2_STA_PB : BOOL ;
   SF_3_LAMP_TEST : BOOL ;
   SF_3_ALARM_ACK : BOOL ;
   SF_3_STA_PB : BOOL ;
   SF_3_STOP_PB : BOOL ;
   SF_3_HIGH_SPEED_SEL : BOOL ;
   SF_3_LOW_SPEED_SEL : BOOL ;
   SF_3_REPAIR_MODE : BOOL ;
   SF_3_MANUAL_MODE : BOOL ;
   SF_3_SEMI_AUTO_MODE : BOOL ;
   SF_3_MACRO_SELECTION : BOOL ;
   SF_3_SPARE_INPUTS : WORD ;
   SF_3_HARD_PROFI_SS : BOOL ;
   LID_LUTTING_TANK_STA_PB : BOOL ;
   LID_LUTTING_TANK_STOP_PB : BOOL ;
   LID_1_MAG_START_PB : BOOL ;
   LID_1_MAG_STOP_PB : BOOL ;
   LID_2_MAG_START_PB : BOOL ;
   LID_2_MAG_STOP_PB : BOOL ;
   LID_3_MAG_START_PB : BOOL ;
   LID_3_MAG_STOP_PB : BOOL ;
   LID_1_OSC_MTR_STA_PB : BOOL ;
   LID_1_OSC_MTR_STOP_PB : BOOL ;
   LID_2_OSC_MTR_STA_PB : BOOL ;
   LID_2_OSC_MTR_STOP_PB : BOOL ;
   LID_3_OSC_MTR_STA_PB : BOOL ;
   LID_3_OSC_MTR_STOP_PB : BOOL ;
   LID_1_FRA_CLRMTR_STA_PB : BOOL ;
   LID_1_FRA_CLRMTR_STOP_PB : BOOL ;
   LID_2_FRA_CLRMTR_STA_PB : BOOL ;
   LID_2_FRA_CLRMTR_STOP_PB : BOOL ;
   LID_3_FRA_CLRMTR_STA_PB : BOOL ;
   LID_3_FRA_CLRMTR_STOP_PB : BOOL ;
   LID_1_CARGE_FWD_STA_PB : BOOL ;	//LID_1_CARGE_FWD_STA_PB
   LID_1_CARGE_REV_STA_PB : BOOL ;	//LID_1_CARGE_REV_STA_PB
   LID_1_VER_UP_STA_PB : BOOL ;	//LID_1_VER_UP_STA_PB
   LID_1_VER_DN_STA_PB : BOOL ;	//LID_1_VER_DN_STA_PB
   LID_1_FRA_CLR_UP_STA : BOOL ;	//LID_1_FRA_CLR_UP_STA
   LID_1_FRA_CLR_DN_STA : BOOL ;	//LID_1_FRA_CLR_DN_STA
   LID_1_TELES_DN_STA : BOOL ;	//LID_1_TELES_DN_STA
   LID_1_TELES_UP_STA : BOOL ;	//LID_1_TELES_UP_STA
   SLIDE_GATE_1_CLOSE_STA : BOOL ;
   SLIDE_GATE_1_OPEN_STA : BOOL ;
   CONTROL_SEL_PB : BOOL ;
   OVEN_CHARGING_PB : BOOL ;
   LT_SF_SELECTION : BOOL ;
   REPAIR_MODE : BOOL ;
   MANUAL_MODE : BOOL ;
   SEMIAUTO_MODE : BOOL ;
   LID_2_CARGE_FWD_STA_PB : BOOL ;	//LID_2_CARGE_FWD_STA_PB
   LID_2_CARGE_REV_STA_PB : BOOL ;	//LID_2_CARGE_REV_STA_PB
   LID_2_VER_UP_STA_PB : BOOL ;	//LID_2_VER_UP_STA_PB
   LID_2_VER_DN_STA_PB : BOOL ;	//LID_2_VER_DN_STA_PB
   LID_2_FRA_CLR_DN_STA : BOOL ;	//LID_2_FRA_CLR_DN_STA
   LID_2_FRA_CLR_UP_STA : BOOL ;	//LID_2_FRA_CLR_UP_STA
   LID_2_TELES_DN_STA : BOOL ;	//LID_2_TELES_DN_STA
   LID_2_TELES_UP_STA : BOOL ;	//LID_2_TELES_UP_STA
   SLIDE_GATE_2_CLOSE_STA : BOOL ;
   SLIDE_GATE_2_OPEN_STA : BOOL ;
   LID_3_CARGE_FWD_STA_PB : BOOL ;	//LID_3_CARGE_FWD_STA_PB
   LID_3_CARGE_REV_STA_PB : BOOL ;	//LID_3_CARGE_REV_STA_PB
   LID_3_FRA_CLR_DN_STA : BOOL ;	//LID_3_FRA_CLR_DN_STA
   LID_3_FRA_CLR_UP_STA : BOOL ;	//LID_3_FRA_CLR_UP_STA
   LID_3_TELES_DN_STA : BOOL ;	//LID_3_TELES_DN_STA
   LID_3_TELES_UP_STA : BOOL ;	//LID_3_TELES_UP_STA
   SLIDE_GATE_3_CLOSE_STA : BOOL ;
   SLIDE_GATE_3_OPEN_STA : BOOL ;
   BUNKER_GATE_START_PB : BOOL ;
   BUNKER_GATE_STOP_PB : BOOL ;
   BNKR_GATE1_CLS_STA_PB : BOOL ;
   BUNKR_GATE1_HME_STA_PB : BOOL ;
   BUNKER_GATE_1_LID1_STOP : BOOL ;
   BNKR_GATE_1_OP_REMODE : BOOL ;
   BNKR_GATE_1_OP_MAN_MODE : BOOL ;
   BUNKR_GAT_CD_SEL : BOOL ;
   BUNKR_GATE1_OPN_STA_PB : BOOL ;
   BNKR_GATE_3_OP_REMODE : BOOL ;
   BNKR_GATE_3_OP_MAN_MODE : BOOL ;
   BUNKR_GAT_3_OP_SAUT_MOD : BOOL ;
   BUNKR_GATE3_OPN_STA_PB : BOOL ;
   BNKR_GATE3_CLS_STA_PB : BOOL ;
   BUNKR_GATE3_HME_STA_PB : BOOL ;
   BUNKER_GATE_3_LID1_STOP : BOOL ;
   PREPARE_TO_CHARGE : BOOL ;
   FINISH_CHARGE_PB : BOOL ;
   LID_1_STOP_PB : BOOL ;
   LID_2_STOP_PB : BOOL ;
   LID_3_STOP_PB : BOOL ;
   SF_1_READY_STA : BOOL ;
   SF_1_RUNNG_FB : BOOL ;
   SF_1_LT_OVEN_CHARGE_STA : BOOL ;
   SF_1_LT_SF_SELECTION : BOOL ;
   AUTO_MODE : BOOL ;
   PUMP1_STA_PB : BOOL ;
   PUMP1_STOP_PB : BOOL ;
   PUMP2_STA_PB : BOOL ;
   PUMP2_STOP_PB : BOOL ;
   START_PB_PUMP_1 : BOOL ;
   STOP_PB_PUMP_1 : BOOL ;
   START_PB_PUMP_2 : BOOL ;
   STOP_PB_PUMP_2 : BOOL ;
   CD_LCS_SELEC1_2_SWITCH : BOOL ;	//CD_LCS_SELEC1_2_SWITCH
   PUMP_SEL_SWITCH_CDL : BOOL ;
   STA_PB_CIR_PUMP : BOOL ;
   STOP_PB_CIR_PUMP : BOOL ;
   STA_PB_COOLER_FAN : BOOL ;
   STOP_PB_COOLER_FAN : BOOL ;
   LAMP_TEST : BOOL ;
   ACCUMULATOR_STA_PB : BOOL ;
   ACCUMULATOR_STOP_PB : BOOL ;
   HEATER_STA_PB : BOOL ;
   SF1_LS_SEL : BOOL ;
   SF1_HS_SEL : BOOL ;
   SPARE : BOOL ;
   SCREW_FEEDER1_STOP_PB : BOOL ;
   SF1_HIGH_SPEED_SEL : BOOL ;
   DRIVE_4_RUNNING_FB : BOOL ;	//SPARE
   SF1_LOW_SPEED_SEL : BOOL ;
   SCREW_FEEDER2_STA_PB : BOOL ;
   SCREW_FEEDER2_STOP_PB : BOOL ;
   SF2_HIGH_SPEED_SEL : BOOL ;
   SF2_LOW_SPEED_SEL : BOOL ;
   SCREW_FEEDER3_STA_PB : BOOL ;
   SCREW_FEEDER3_STOP_PB : BOOL ;
   SF3_HIGH_SPEED_SEL : BOOL ;
   SF3_LOW_SPEED_SEL : BOOL ;
   LID_LUT_TANK_READY_FB : BOOL ;	//LID LUTTING TANK READY FOR START
   LID_LUTTING_TANK_RUN_FB : BOOL ;	//LID LUTTING TANK RUNNING FB
   LID_LUT_TANK_OLR_TRIP : BOOL ;	//LID LUTTING TANK OLR TRIP
   LID_LUTTING_TANK_STAR_PB : BOOL ;	//LID LUTTING TANK START PB
   STAT_1 : BOOL ;	//LID LUTTING TANK STOP PB
   LID_MECHANIS_REP_MODE : BOOL ;
   LID_MECHANIS_MAN_MODE : BOOL ;
   LID_MECH_SEMI_AUT_MODE : BOOL ;
   LID_FR_CLNR_AUTO_MODE : BOOL ;	//SPARE
   CDC_EMERGENCY : BOOL ;	//CDC_EMERGENCY
   B_GATE_COAL_LOD_STA_PB : BOOL ;	//B_GATE_COAL_LOD_STP_PB
   B_GATE_COAL_LOD_STP_PB : BOOL ;	//B_GATE_COAL_LOD_STA_PB
   LID_FRAME_CLR_BYBASS : BOOL ;	//LID_FRAME_CLR_BYBASS
   AUTO_POSITION_ACK : BOOL ;	//SPARE
   HOPPER_STOP_PB : BOOL ;	//SPARE
   LID_LUTTING_STA_PB : BOOL ;	//SPARE
   BG_1_UP_STA_PB_CD : BOOL ;
   BG_1_DOWN_STA_PB_CD : BOOL ;
   BG_1_DOWN_STA_PB_CD_2 : BOOL ;
   BG_3_UP_STA_PB_CD : BOOL ;
   BG_3_DOWN_STA_PB_CD : BOOL ;
   BG_3_DOWN_STA_PB_CD_2 : BOOL ;
   LASER_SPOTTING : BOOL ;
   LAMP_TEST_1 : BOOL ;
   LID_3_VER_DN_STA_PB : BOOL ;
   BNKR_GATE2_UP_STA_PB : BOOL ;
   BNKR_GATE2_DNSTAPB : BOOL ;
   BNKR_GATE_2_OP_STA_PB_CD : BOOL ;
   BNKR_GATE_2_CL_STA_PB : BOOL ;
   BUN_GATE_2_HOME_STA_PB : BOOL ;
   LID_LIFTR3_VER_UP_START : BOOL ;
   SF_2_LOW_SPD_SEL : BOOL ;
   SF_2_HIGH_SPD_SEL : BOOL ;
   EMER_STOP_CD : BOOL ;
   QQ : BOOL ;
   WW : BOOL ;
   EE : BOOL ;
   AA : BOOL ;
   MAN_REPAIR_SELECTOR : BOOL ;
   QQ1 : BOOL ;
   QQ2 : BOOL ;
   WW1 : BOOL ;
   EE1 : BOOL ;
   AA1 : BOOL ;
   AA11 : BOOL ;
   AA111 : BOOL ;
   AUTO_SELECTOR_SWITCH : BOOL ;
   QQ11 : BOOL ;
   QQ21 : BOOL ;
   WW11 : BOOL ;
   EE11 : BOOL ;
   AA12 : BOOL ;
   AA112 : BOOL ;
   AA1111 : BOOL ;
   PUMP_SELECTOR_SW : BOOL ;
   QQ3 : BOOL ;
   WW2 : BOOL ;
   EE2 : BOOL ;
   AA2 : BOOL ;
   QQ12 : BOOL ;
   QQ22 : BOOL ;
   WW12 : BOOL ;
   CD_LCS_SELECTOR : BOOL ;
   QQ31 : BOOL ;
   WW21 : BOOL ;
   EE21 : BOOL ;
   AA21 : BOOL ;
   QQ121 : BOOL ;
   QQ221 : BOOL ;
   WW121 : BOOL ;
   CD_LCS_1_2_SS : BOOL ;
   QQ111 : BOOL ;
   QQ211 : BOOL ;
   WW111 : BOOL ;
   EE111 : BOOL ;
   AA121 : BOOL ;
   AA1121 : BOOL ;
   AA11111 : BOOL ;
   HIGH_LOW_SPD_SF_1 : BOOL ;
   A : BOOL ;
   QQ2111 : BOOL ;
   WW1111 : BOOL ;
   EE1111 : BOOL ;
   AA1211 : BOOL ;
   AA11211 : BOOL ;
   AA111111 : BOOL ;
   HIGH_LOW_SPD_SF_2 : BOOL ;
   A1 : BOOL ;
   QQ21111 : BOOL ;
   WW11111 : BOOL ;
   EE11111 : BOOL ;
   AA12111 : BOOL ;
   AA112111 : BOOL ;
   AA1111111 : BOOL ;
   HIGH_LOW_SPD_SF_3 : BOOL ;
   A11 : BOOL ;
   QQ211111 : BOOL ;
   WW111111 : BOOL ;
   EE111111 : BOOL ;
   AA121111 : BOOL ;
   AA1121111 : BOOL ;
   AA11111111 : BOOL ;
   OPER_MODE : BOOL ;
   QQ2111111 : BOOL ;
   WW1111111 : BOOL ;
   EE1111111 : BOOL ;
   AA1211111 : BOOL ;
   AA11211111 : BOOL ;
   AA111111111 : BOOL ;
   QSA : BOOL ;
   LID_FRM_CLNR_BYPASS_SS : BOOL ;
   A111 : BOOL ;
   QQ2111112 : BOOL ;
   WW1111112 : BOOL ;
   EE1111112 : BOOL ;
   AA1211112 : BOOL ;
   AA11211112 : BOOL ;
   AA111111112 : BOOL ;
   LID_FRAME_BYPASS : BOOL ;
   A1111 : BOOL ;
   QQ21111121 : BOOL ;
   WW11111121 : BOOL ;
   EE11111121 : BOOL ;
   AA12111121 : BOOL ;
   AA112111121 : BOOL ;
   AA1111111121 : BOOL ;
   BUNKER_GATE_CD_LCS_SS : BOOL ;
   QQ21111111 : BOOL ;
   WW11111111 : BOOL ;
   EE11111111 : BOOL ;
   AA12111111 : BOOL ;
   AA112111111 : BOOL ;
   AA1111111111 : BOOL ;
   QSA1 : BOOL ;
   TRAV_AUTO_MAN_SS : BOOL ;
   QQ211111111 : BOOL ;
   WW111111111 : BOOL ;
   EE111111111 : BOOL ;
   AA121111111 : BOOL ;
   AA1121111111 : BOOL ;
   AA11111111111 : BOOL ;
   QSA11 : BOOL ;
   TRAV_AUTO_MAN_SELEC : BOOL ;
   NO_USE : BOOL ;
   NO_USE1 : BOOL ;
   NO_USE2 : BOOL ;
   NO_USE3 : BOOL ;
   NO_USE4 : BOOL ;
   NO_USE5 : BOOL ;
   NO_USE6 : BOOL ;
  END_STRUCT ;	
BEGIN
END_DATA_BLOCK

DATA_BLOCK "SCREW_FEEDER_PF"	// DB 17
VERSION : 0.1
  STRUCT
   SF1_REF_WITH_LIMIT : BOOL ;	//SCREW FEEDER-1 RESERVED1 BIT
   SF1_LOCAL_REMOTE_BI : BOOL ;	//SCREW FEEDER-1 PROFIBUS SELECTED BIT
   SF1_ACT_ABOVE_LMIT : BOOL ;	//SCREW FEEDER-1 REFERENCE REACHED BIT
   SF1_PROFI_SELECTED : BOOL ;	//SCREW FEEDER-1 RESERVED2 BIT
   SF1_EXTRNL_RUN_BIT : BOOL ;	//SCREW FEEDER-1 RESERVED3 BIT
   SF1_RESERVED1_BIT : BOOL ;	//SCREW FEEDER-1 RESERVED4 BIT
   SF1_RESERVED2_BIT : BOOL ;	//SCREW FEEDER-1 RESERVED5 BIT
   SF1_RESERVED3_BIT : BOOL ;	//SCREW FEEDER-1 REVERSE DIRECTION BIT
   SF1_RDY_SWITCH_ON : BOOL ;	//SCREW FEEDER-1 READY TO SWITCH ON BIT
   SF1_RDY_BIT : BOOL ;	//SCREW FEEDER-1 READY BIT
   SF1_RUNNING_BIT : BOOL ;	//SCREW FEEDER-1 RUNNING BIT
   SF1_FAULT_BIT : BOOL ;	//SCREW FEEDER-1 FAULT BIT
   SF1_OFF2_BIT : BOOL ;	//SCREW FEEDER-1 VOLTAGE ENABLED BIT
   SF1_OFF3_BIT : BOOL ;	//SCREW FEEDER-1 EMERGENCY STOP BIT
   SF1_SWTCHON_DISABLE : BOOL ;	//SCREW FEEDER-1 SWITCH ON DISABLE BIT
   SF1_ALARM_BIT : BOOL ;	//SCREW FEEDER-1 ALARM BIT
   SF1_SPEED_ACTUAL : INT ;	//SCREW FEEDER-1 SPEED ACTUAL VALUE
   SF1_CONTROLWORD : WORD ;	//SCREW FEEDER-1 CONTROL WORD VALUE
   SF1_SPEED_REF : INT ;	//SCREW FEEDER-1 SPEED REFERENCE VALUE
   SF2_REF_WITH_LIMIT1 : BOOL ;	//SCREW FEEDER-2 RESERVED1 BIT
   SF2_LOCAL_REMOTE_BI : BOOL ;	//SCREW FEEDER-2 PROFIBUS SELECTED BIT
   SF2_ACT_ABOVE_LMIT : BOOL ;	//SCREW FEEDER-2 REFERENCE REACHED BIT
   SF2_PROFI_SELECTED : BOOL ;	//SCREW FEEDER-2 RESERVED2 BIT
   SF2_EXTRNL_RUN_BIT : BOOL ;	//SCREW FEEDER-2 RESERVED3 BIT
   SF2_RESERVED1_BIT : BOOL ;	//SCREW FEEDER-2 RESERVED4 BIT
   SF2_RESERVED2_BIT : BOOL ;	//SCREW FEEDER-2 RESERVED5 BIT
   SF2_RESERVED3_BIT : BOOL ;	//SCREW FEEDER-2 REVERSE DIRECTION BIT
   SF2_RDY_SWITCH_ON : BOOL ;	//SCREW FEEDER-2 READY TO SWITCH ON BIT
   SF2_RDY_BIT : BOOL ;	//SCREW FEEDER-2 READY BIT
   SF2_RUNNING_BIT : BOOL ;	//SCREW FEEDER-2 RUNNING BIT
   SF2_FAULT_BIT : BOOL ;	//SCREW FEEDER-2 FAULT BIT
   SF2_OFF2_BIT : BOOL ;	//SCREW FEEDER-2 VOLTAGE ENABLED BIT
   SF2_OFF3_BIT : BOOL ;	//SCREW FEEDER-2 EMERGENCY STOP BIT
   SF2_SWTCHON_DISABLE : BOOL ;	//SCREW FEEDER-2 SWITCH ON DISABLE BIT
   SF2_ALARM_BIT : BOOL ;	//SCREW FEEDER-2 ALARM BIT
   SF2_SPEED_ACTUAL : INT ;	//SCREW FEEDER-2 SPEED ACTUAL VALUE
   SF2_CONTROLWORD : WORD ;	//SCREW FEEDER-2 CONTROL WORD VALUE
   SF2_SPEED_REF : INT ;	//SCREW FEEDER-2 SPEED REFERENCE VALUE
   SF3_REF_WITH_LIMIT : BOOL ;	//SCREW FEEDER-3 RESERVED1 BIT
   SF3_LOCAL_REMOTE_BIT : BOOL ;	//SCREW FEEDER-3 PROFIBUS SELECTED BIT
   SF3_ACT_ABOVE_LMIT : BOOL ;	//SCREW FEEDER-3 REFERENCE REACHED BIT
   SF3_PROFI_SELECTED : BOOL ;	//SCREW FEEDER-3 RESERVED2 BIT
   SF3_EXTRNL_RUN_BIT : BOOL ;	//SCREW FEEDER-3 RESERVED3 BIT
   SF3_RESERVED1_BIT : BOOL ;	//SCREW FEEDER-3 RESERVED4 BIT
   SF3_RESERVED2_BIT : BOOL ;	//SCREW FEEDER-3 RESERVED5 BIT
   SF3_RESERVED3_BIT : BOOL ;	//SCREW FEEDER-3 REVERSE DIRECTION BIT
   SF3_RDY_SWITCH_ON : BOOL ;	//SCREW FEEDER-3 READY TO SWITCH ON BIT
   SF3_RDY_BIT : BOOL ;	//SCREW FEEDER-3 READY BIT
   SF3_RUNNING_BIT : BOOL ;	//SCREW FEEDER-3 RUNNING BIT
   SF3_FAULT_BIT : BOOL ;	//SCREW FEEDER-3 FAULT BIT
   SF3_OFF2_BIT : BOOL ;	//SCREW FEEDER-3 VOLTAGE ENABLED BIT
   SF3_OFF3_BIT : BOOL ;	//SCREW FEEDER-3 EMERGENCY STOP BIT
   SF3_SWTCHON_DISABLE : BOOL ;	//SCREW FEEDER-3 SWITCH ON DISABLE BIT
   SF3_ALARM_BIT : BOOL ;	//SCREW FEEDER-3 ALARM BIT
   SF3_SPEED_ACTUAL : INT ;	//SCREW FEEDER-3 SPEED ACTUAL VALUE
   SF3_CONTROLWORD : WORD ;	//SCREW FEEDER-3 CONTROL WORD VALUE
   SF3_SPEED_REF : INT ;	//SCREW FEEDER-3 SPEED REFERENCE VALUE
  END_STRUCT ;	
BEGIN
END_DATA_BLOCK

